(* Logix 5000 project; controller reports 1756-L63 rev 20.15; software revision 20.04; part 37 of 52 *)

        [52].log_data[51].valid := 1, [52].log_data[52].min := -1.6399994, [52].log_data[52].max := -1.4800034, [52].log_data[52].total := -5567.262, [52].log_data[52].time := 3600.0, [52].log_data[52].minminute := 39, [52].log_data[52].valid := 1, [52].log_data[53].min := -1.5600052, [52].log_data[53].max := -1.4199982, [52].log_data[53].total := -5304.3613, [52].log_data[53].time := 3600.0, [52].log_data[53].minminute := 16, [52].log_data[53].valid := 1, [52].log_data[54].time := 3600.0, [52].log_data[54].valid := 1, [52].log_data[55].time := 3600.0, [52].log_data[55].valid := 1, [52].log_data[56].min := 0.16024561, [52].log_data[56].max := 0.16063818, [52].log_data[56].total := 577.39246, [52].log_data[56].time := 3600.0, [52].log_data[56].minminute := 9, [52].log_data[56].valid := 1, [52].log_data[57].min := 0.27864859, [52].log_data[57].max := 0.27904117, [52].log_data[57].total := 1003.6821, [52].log_data[57].time := 3600.0, [52].log_data[57].minminute := 10, [52].log_data[57].maxminute := 2, [52].log_data[57].valid := 1, [52].log_data[58].time := 3600.0, [52].log_data[58].valid := 1, [52].log_data[59].time := 3600.0, [52].log_data[59].valid := 1, [52].log_data[60].valid := 1, [52].log_data[61].valid := 1, [52].log_data[62].valid := 1, [52].log_data[63].valid := 1, [52].log_data[64].valid := 1, [52].log_data[65].valid := 1, [52].log_data[66].valid := 1, [52].log_data[67].valid := 1, [52].log_data[68].valid := 1, [52].log_data[69].valid := 1, [52].log_data[70].valid := 1, [52].log_data[71].valid := 1, [52].log_data[72].valid := 1, [52].log_data[73].valid := 1, [52].log_data[74].valid := 1, [52].log_data[75].valid := 1, [52].log_data[76].valid := 1, [52].log_data[77].valid := 1, [52].log_data[78].valid := 1, [52].log_data[79].valid := 1, [52].log_data[80].valid := 1, [52].log_data[81].valid := 1, [52].log_data[82].valid := 1, [52].log_data[83].valid := 1, [52].log_data[84].valid := 1, [52].log_data[85].valid := 1,
        [52].log_data[86].valid := 1, [52].log_data[87].valid := 1, [52].log_data[88].valid := 1, [52].log_data[89].valid := 1, [52].log_data[90].valid := 1, [52].log_data[91].valid := 1, [52].log_data[92].valid := 1, [52].log_data[93].valid := 1, [52].log_data[94].valid := 1, [52].log_data[95].valid := 1, [52].log_data[96].valid := 1, [52].log_data[97].valid := 1, [52].log_data[98].valid := 1, [52].log_data[99].valid := 1, [52].log_data[100].valid := 1, [52].log_data[101].valid := 1, [52].log_data[102].valid := 1, [52].log_data[103].valid := 1, [52].log_data[104].valid := 1, [52].log_data[105].valid := 1, [52].log_data[106].valid := 1, [52].log_data[107].valid := 1, [52].log_data[108].valid := 1, [52].log_data[109].valid := 1, [52].log_data[110].valid := 1, [52].log_data[111].valid := 1, [52].log_data[112].valid := 1, [52].log_data[113].valid := 1, [52].log_data[114].valid := 1, [52].log_data[115].valid := 1, [52].log_data[116].valid := 1, [52].log_data[117].valid := 1, [52].log_data[118].valid := 1, [52].log_data[119].valid := 1, [52].log_data[120].valid := 1, [52].log_data[121].valid := 1, [52].log_data[122].valid := 1, [52].log_data[123].valid := 1, [52].log_data[124].valid := 1, [52].time.Year := 2023, [52].time.Month := 1, [52].time.Day := 15, [52].time.Hour := 7, [52].time.Minute := 59, [52].time.Second := 59, [53].log_data[0].min := 1.0, [53].log_data[0].max := 1.0, [53].log_data[0].total := 3600.0, [53].log_data[0].time := 3600.0, [53].log_data[0].valid := 1, [53].log_data[1].max := 1.0, [53].log_data[1].total := 543.5, [53].log_data[1].time := 3600.0, [53].log_data[1].maxminute := 32, [53].log_data[1].valid := 1, [53].log_data[2].max := 1.0, [53].log_data[2].total := 540.0, [53].log_data[2].time := 3600.0, [53].log_data[2].maxminute := 32, [53].log_data[2].valid := 1,
        [53].log_data[3].time := 3600.0, [53].log_data[3].valid := 1, [53].log_data[4].time := 3600.0, [53].log_data[4].valid := 1, [53].log_data[5].max := 1.0, [53].log_data[5].total := 221.5, [53].log_data[5].time := 3600.0, [53].log_data[5].maxminute := 33, [53].log_data[5].valid := 1, [53].log_data[6].time := 3600.0, [53].log_data[6].valid := 1, [53].log_data[7].time := 3600.0, [53].log_data[7].valid := 1, [53].log_data[8].max := 1.0, [53].log_data[8].total := 1510.749, [53].log_data[8].time := 3600.0, [53].log_data[8].maxminute := 34, [53].log_data[8].valid := 1, [53].log_data[9].max := 1.0, [53].log_data[9].total := 1507.249, [53].log_data[9].time := 3600.0, [53].log_data[9].maxminute := 34, [53].log_data[9].valid := 1, [53].log_data[10].min := 1.0, [53].log_data[10].max := 1.0, [53].log_data[10].total := 3600.0, [53].log_data[10].time := 3600.0, [53].log_data[10].valid := 1, [53].log_data[11].time := 3600.0, [53].log_data[11].valid := 1, [53].log_data[12].min := 1.0, [53].log_data[12].max := 1.0, [53].log_data[12].total := 3600.0, [53].log_data[12].time := 3600.0, [53].log_data[12].valid := 1, [53].log_data[13].min := 1.0, [53].log_data[13].max := 1.0, [53].log_data[13].total := 3600.0, [53].log_data[13].time := 3600.0, [53].log_data[13].valid := 1, [53].log_data[14].time := 3600.0, [53].log_data[14].valid := 1, [53].log_data[15].time := 3600.0, [53].log_data[15].valid := 1, [53].log_data[16].time := 3600.0, [53].log_data[16].valid := 1, [53].log_data[17].min := 1.0, [53].log_data[17].max := 1.0, [53].log_data[17].total := 3600.0, [53].log_data[17].time := 3600.0, [53].log_data[17].valid := 1, [53].log_data[18].time := 3600.0, [53].log_data[18].valid := 1, [53].log_data[19].time := 3600.0, [53].log_data[19].valid := 1, [53].log_data[20].time := 3600.0, [53].log_data[20].valid := 1, [53].log_data[21].min := 1.0, [53].log_data[21].max := 1.0, [53].log_data[21].total := 3600.0,
        [53].log_data[21].time := 3600.0, [53].log_data[21].valid := 1, [53].log_data[22].time := 3600.0, [53].log_data[22].valid := 1, [53].log_data[23].time := 3600.0, [53].log_data[23].valid := 1, [53].log_data[24].time := 3600.0, [53].log_data[24].valid := 1, [53].log_data[25].time := 3600.0, [53].log_data[25].valid := 1, [53].log_data[26].time := 3600.0, [53].log_data[26].valid := 1, [53].log_data[27].time := 3600.0, [53].log_data[27].valid := 1, [53].log_data[28].time := 3600.0, [53].log_data[28].valid := 1, [53].log_data[29].min := 1.0, [53].log_data[29].max := 1.0, [53].log_data[29].total := 3600.0, [53].log_data[29].time := 3600.0, [53].log_data[29].valid := 1, [53].log_data[30].min := 1.0, [53].log_data[30].max := 1.0, [53].log_data[30].total := 3600.0, [53].log_data[30].time := 3600.0, [53].log_data[30].valid := 1, [53].log_data[31].max := 1.0, [53].log_data[31].total := 543.249, [53].log_data[31].time := 3600.0, [53].log_data[31].maxminute := 43, [53].log_data[31].valid := 1, [53].log_data[32].max := 1.0, [53].log_data[32].total := 783.998, [53].log_data[32].time := 3600.0, [53].log_data[32].maxminute := 34, [53].log_data[32].valid := 1, [53].log_data[33].time := 3600.0, [53].log_data[33].valid := 1, [53].log_data[34].time := 3600.0, [53].log_data[34].valid := 1, [53].log_data[35].max := 1.0, [53].log_data[35].total := 640.49805, [53].log_data[35].time := 3600.0, [53].log_data[35].maxminute := 37, [53].log_data[35].valid := 1, [53].log_data[36].max := 1.0, [53].log_data[36].total := 594.998, [53].log_data[36].time := 3600.0, [53].log_data[36].maxminute := 34, [53].log_data[36].valid := 1, [53].log_data[37].max := 7.248974, [53].log_data[37].total := 3411.01, [53].log_data[37].time := 3600.0, [53].log_data[37].maxminute := 33, [53].log_data[37].valid := 1, [53].log_data[38].time := 3600.0, [53].log_data[38].valid := 1, [53].log_data[39].min := 0.99788606, [53].log_data[39].max := 1.0216767, [53].log_data[39].total := 3646.9153,
        [53].log_data[39].time := 3600.0, [53].log_data[39].minminute := 35, [53].log_data[39].maxminute := 37, [53].log_data[39].valid := 1, [53].log_data[40].min := 7.5687137, [53].log_data[40].max := 7.6019654, [53].log_data[40].total := 27316.076, [53].log_data[40].time := 3600.0, [53].log_data[40].minminute := 7, [53].log_data[40].maxminute := 11, [53].log_data[40].valid := 1, [53].log_data[41].min := 0.025680907, [53].log_data[41].max := 0.045309816, [53].log_data[41].total := 128.45833, [53].log_data[41].time := 3600.0, [53].log_data[41].minminute := 59, [53].log_data[41].maxminute := 29, [53].log_data[41].valid := 1, [53].log_data[42].min := 2.2918782, [53].log_data[42].max := 2.296707, [53].log_data[42].total := 8260.53, [53].log_data[42].time := 3600.0, [53].log_data[42].minminute := 43, [53].log_data[42].maxminute := 41, [53].log_data[42].valid := 1, [53].log_data[43].min := -0.27999878, [53].log_data[43].max := -0.26000214, [53].log_data[43].total := -988.176, [53].log_data[43].time := 3600.0, [53].log_data[43].valid := 1, [53].log_data[44].min := -0.30000305, [53].log_data[44].max := -0.30000305, [53].log_data[44].total := -1080.0911, [53].log_data[44].time := 3600.0, [53].log_data[44].valid := 1, [53].log_data[45].time := 3600.0, [53].log_data[45].valid := 1, [53].log_data[46].time := 3600.0, [53].log_data[46].valid := 1, [53].log_data[47].time := 3600.0, [53].log_data[47].valid := 1, [53].log_data[48].min := 6.6066113, [53].log_data[48].max := 6.9619374, [53].log_data[48].total := 24341.145, [53].log_data[48].time := 3600.0, [53].log_data[48].minminute := 59, [53].log_data[48].maxminute := 39, [53].log_data[48].valid := 1, [53].log_data[49].min := 7.224471, [53].log_data[49].max := 9.765266, [53].log_data[49].total := 32563.492, [53].log_data[49].time := 3600.0, [53].log_data[49].minminute := 55, [53].log_data[49].maxminute := 20, [53].log_data[49].valid := 1, [53].log_data[50].min := 2.061275, [53].log_data[50].max := 2.150784, [53].log_data[50].total := 7565.2534, [53].log_data[50].time := 3600.0, [53].log_data[50].minminute := 37,
        [53].log_data[50].maxminute := 34, [53].log_data[50].valid := 1, [53].log_data[51].time := 3600.0, [53].log_data[51].valid := 1, [53].log_data[52].min := -4.3799973, [53].log_data[52].max := 0.11999512, [53].log_data[52].total := -6630.809, [53].log_data[52].time := 3600.0, [53].log_data[52].minminute := 35, [53].log_data[52].maxminute := 41, [53].log_data[52].valid := 1, [53].log_data[53].min := -3.9399948, [53].log_data[53].max := 0.27999878, [53].log_data[53].total := -5923.6562, [53].log_data[53].time := 3600.0, [53].log_data[53].minminute := 35, [53].log_data[53].maxminute := 58, [53].log_data[53].valid := 1, [53].log_data[54].max := 0.5165, [53].log_data[54].total := 524.9467, [53].log_data[54].time := 3600.0, [53].log_data[54].maxminute := 35, [53].log_data[54].valid := 1, [53].log_data[55].max := 0.5265, [53].log_data[55].total := 486.45926, [53].log_data[55].time := 3600.0, [53].log_data[55].maxminute := 58, [53].log_data[55].valid := 1, [53].log_data[56].min := 0.16016708, [53].log_data[56].max := 0.16059892, [53].log_data[56].total := 577.3497, [53].log_data[56].time := 3600.0, [53].log_data[56].minminute := 43, [53].log_data[56].maxminute := 5, [53].log_data[56].valid := 1, [53].log_data[57].min := 0.27860934, [53].log_data[57].max := 0.27904117, [53].log_data[57].total := 1003.57135, [53].log_data[57].time := 3600.0, [53].log_data[57].minminute := 7, [53].log_data[57].maxminute := 13, [53].log_data[57].valid := 1, [53].log_data[58].time := 3600.0, [53].log_data[58].valid := 1, [53].log_data[59].time := 3600.0, [53].log_data[59].valid := 1, [53].log_data[60].valid := 1, [53].log_data[61].valid := 1, [53].log_data[62].valid := 1, [53].log_data[63].valid := 1, [53].log_data[64].valid := 1, [53].log_data[65].valid := 1, [53].log_data[66].valid := 1, [53].log_data[67].valid := 1, [53].log_data[68].valid := 1, [53].log_data[69].valid := 1, [53].log_data[70].valid := 1, [53].log_data[71].valid := 1, [53].log_data[72].valid := 1, [53].log_data[73].valid := 1,
        [53].log_data[74].valid := 1, [53].log_data[75].valid := 1, [53].log_data[76].valid := 1, [53].log_data[77].valid := 1, [53].log_data[78].valid := 1, [53].log_data[79].valid := 1, [53].log_data[80].valid := 1, [53].log_data[81].valid := 1, [53].log_data[82].valid := 1, [53].log_data[83].valid := 1, [53].log_data[84].valid := 1, [53].log_data[85].valid := 1, [53].log_data[86].valid := 1, [53].log_data[87].valid := 1, [53].log_data[88].valid := 1, [53].log_data[89].valid := 1, [53].log_data[90].valid := 1, [53].log_data[91].valid := 1, [53].log_data[92].valid := 1, [53].log_data[93].valid := 1, [53].log_data[94].valid := 1, [53].log_data[95].valid := 1, [53].log_data[96].valid := 1, [53].log_data[97].valid := 1, [53].log_data[98].valid := 1, [53].log_data[99].valid := 1, [53].log_data[100].valid := 1, [53].log_data[101].valid := 1, [53].log_data[102].valid := 1, [53].log_data[103].valid := 1, [53].log_data[104].valid := 1, [53].log_data[105].valid := 1, [53].log_data[106].valid := 1, [53].log_data[107].valid := 1, [53].log_data[108].valid := 1, [53].log_data[109].valid := 1, [53].log_data[110].valid := 1, [53].log_data[111].valid := 1, [53].log_data[112].valid := 1, [53].log_data[113].valid := 1, [53].log_data[114].valid := 1, [53].log_data[115].valid := 1, [53].log_data[116].valid := 1, [53].log_data[117].valid := 1, [53].log_data[118].valid := 1, [53].log_data[119].valid := 1, [53].log_data[120].valid := 1, [53].log_data[121].valid := 1, [53].log_data[122].valid := 1, [53].log_data[123].valid := 1, [53].log_data[124].valid := 1, [53].time.Year := 2023, [53].time.Month := 1, [53].time.Day := 15, [53].time.Hour := 8, [53].time.Minute := 59, [53].time.Second := 59, [54].log_data[0].min := 1.0, [54].log_data[0].max := 1.0, [54].log_data[0].total := 3600.0,
        [54].log_data[0].time := 3600.0, [54].log_data[0].valid := 1, [54].log_data[1].time := 3600.0, [54].log_data[1].valid := 1, [54].log_data[2].time := 3600.0, [54].log_data[2].valid := 1, [54].log_data[3].time := 3600.0, [54].log_data[3].valid := 1, [54].log_data[4].time := 3600.0, [54].log_data[4].valid := 1, [54].log_data[5].max := 1.0, [54].log_data[5].total := 46.5, [54].log_data[5].time := 3600.0, [54].log_data[5].maxminute := 2, [54].log_data[5].valid := 1, [54].log_data[6].time := 3600.0, [54].log_data[6].valid := 1, [54].log_data[7].time := 3600.0, [54].log_data[7].valid := 1, [54].log_data[8].min := 1.0, [54].log_data[8].max := 1.0, [54].log_data[8].total := 3600.0, [54].log_data[8].time := 3600.0, [54].log_data[8].valid := 1, [54].log_data[9].min := 1.0, [54].log_data[9].max := 1.0, [54].log_data[9].total := 3600.0, [54].log_data[9].time := 3600.0, [54].log_data[9].valid := 1, [54].log_data[10].min := 1.0, [54].log_data[10].max := 1.0, [54].log_data[10].total := 3600.0, [54].log_data[10].time := 3600.0, [54].log_data[10].valid := 1, [54].log_data[11].time := 3600.0, [54].log_data[11].valid := 1, [54].log_data[12].min := 1.0, [54].log_data[12].max := 1.0, [54].log_data[12].total := 3600.0, [54].log_data[12].time := 3600.0, [54].log_data[12].valid := 1, [54].log_data[13].min := 1.0, [54].log_data[13].max := 1.0, [54].log_data[13].total := 3600.0, [54].log_data[13].time := 3600.0, [54].log_data[13].valid := 1, [54].log_data[14].time := 3600.0, [54].log_data[14].valid := 1, [54].log_data[15].time := 3600.0, [54].log_data[15].valid := 1, [54].log_data[16].time := 3600.0, [54].log_data[16].valid := 1, [54].log_data[17].min := 1.0, [54].log_data[17].max := 1.0, [54].log_data[17].total := 3600.0, [54].log_data[17].time := 3600.0, [54].log_data[17].valid := 1, [54].log_data[18].time := 3600.0, [54].log_data[18].valid := 1, [54].log_data[19].time := 3600.0,
        [54].log_data[19].valid := 1, [54].log_data[20].time := 3600.0, [54].log_data[20].valid := 1, [54].log_data[21].min := 1.0, [54].log_data[21].max := 1.0, [54].log_data[21].total := 3600.0, [54].log_data[21].time := 3600.0, [54].log_data[21].valid := 1, [54].log_data[22].time := 3600.0, [54].log_data[22].valid := 1, [54].log_data[23].time := 3600.0, [54].log_data[23].valid := 1, [54].log_data[24].time := 3600.0, [54].log_data[24].valid := 1, [54].log_data[25].time := 3600.0, [54].log_data[25].valid := 1, [54].log_data[26].time := 3600.0, [54].log_data[26].valid := 1, [54].log_data[27].time := 3600.0, [54].log_data[27].valid := 1, [54].log_data[28].time := 3600.0, [54].log_data[28].valid := 1, [54].log_data[29].min := 1.0, [54].log_data[29].max := 1.0, [54].log_data[29].total := 3600.0, [54].log_data[29].time := 3600.0, [54].log_data[29].valid := 1, [54].log_data[30].min := 1.0, [54].log_data[30].max := 1.0, [54].log_data[30].total := 3600.0, [54].log_data[30].time := 3600.0, [54].log_data[30].valid := 1, [54].log_data[31].max := 1.0, [54].log_data[31].total := 1629.998, [54].log_data[31].time := 3600.0, [54].log_data[31].maxminute := 4, [54].log_data[31].valid := 1, [54].log_data[32].max := 1.0, [54].log_data[32].total := 1440.498, [54].log_data[32].time := 3600.0, [54].log_data[32].minminute := 2, [54].log_data[32].valid := 1, [54].log_data[33].time := 3600.0, [54].log_data[33].valid := 1, [54].log_data[34].time := 3600.0, [54].log_data[34].valid := 1, [54].log_data[35].max := 1.0, [54].log_data[35].total := 1532.249, [54].log_data[35].time := 3600.0, [54].log_data[35].minminute := 7, [54].log_data[35].valid := 1, [54].log_data[36].max := 1.0, [54].log_data[36].total := 1626.2471, [54].log_data[36].time := 3600.0, [54].log_data[36].maxminute := 8, [54].log_data[36].valid := 1, [54].log_data[37].time := 3600.0, [54].log_data[37].valid := 1, [54].log_data[38].time := 3600.0, [54].log_data[38].valid := 1,
        [54].log_data[39].min := 0.9956484, [54].log_data[39].max := 1.0202634, [54].log_data[39].total := 3613.4626, [54].log_data[39].time := 3600.0, [54].log_data[39].minminute := 15, [54].log_data[39].maxminute := 2, [54].log_data[39].valid := 1, [54].log_data[40].min := 7.561569, [54].log_data[40].max := 7.603339, [54].log_data[40].total := 27314.873, [54].log_data[40].time := 3600.0, [54].log_data[40].minminute := 48, [54].log_data[40].maxminute := 51, [54].log_data[40].valid := 1, [54].log_data[41].min := 0.022540038, [54].log_data[41].max := 0.03628052, [54].log_data[41].total := 103.08068, [54].log_data[41].time := 3600.0, [54].log_data[41].minminute := 3, [54].log_data[41].maxminute := 37, [54].log_data[41].valid := 1, [54].log_data[42].min := 2.2918782, [54].log_data[42].max := 2.296707, [54].log_data[42].total := 8260.271, [54].log_data[42].time := 3600.0, [54].log_data[42].minminute := 30, [54].log_data[42].maxminute := 36, [54].log_data[42].valid := 1, [54].log_data[43].min := -0.27999878, [54].log_data[43].max := -0.26000214, [54].log_data[43].total := -958.51483, [54].log_data[43].time := 3600.0, [54].log_data[43].valid := 1, [54].log_data[44].min := -0.30000305, [54].log_data[44].max := -0.27999878, [54].log_data[44].total := -1075.2991, [54].log_data[44].time := 3600.0, [54].log_data[44].maxminute := 35, [54].log_data[44].valid := 1, [54].log_data[45].time := 3600.0, [54].log_data[45].valid := 1, [54].log_data[46].time := 3600.0, [54].log_data[46].valid := 1, [54].log_data[47].time := 3600.0, [54].log_data[47].valid := 1, [54].log_data[48].min := 6.585176, [54].log_data[48].max := 6.8080454, [54].log_data[48].total := 24163.797, [54].log_data[48].time := 3600.0, [54].log_data[48].minminute := 2, [54].log_data[48].maxminute := 3, [54].log_data[48].valid := 1, [54].log_data[49].min := 7.171669, [54].log_data[49].max := 9.702061, [54].log_data[49].total := 31267.357, [54].log_data[49].time := 3600.0, [54].log_data[49].minminute := 7, [54].log_data[49].maxminute := 59, [54].log_data[49].valid := 1, [54].log_data[50].min := 2.0161674,
        [54].log_data[50].max := 2.0949588, [54].log_data[50].total := 7409.2114, [54].log_data[50].time := 3600.0, [54].log_data[50].minminute := 59, [54].log_data[50].maxminute := 4, [54].log_data[50].valid := 1, [54].log_data[51].time := 3600.0, [54].log_data[51].valid := 1, [54].log_data[52].min := -2.9400024, [54].log_data[52].max := 0.11999512, [54].log_data[52].total := -7493.728, [54].log_data[52].time := 3600.0, [54].log_data[52].minminute := 25, [54].log_data[52].maxminute := 2, [54].log_data[52].valid := 1, [54].log_data[53].min := -2.5, [54].log_data[53].max := 0.22000122, [54].log_data[53].total := -7034.502, [54].log_data[53].time := 3600.0, [54].log_data[53].minminute := 19, [54].log_data[53].maxminute := 8, [54].log_data[53].valid := 1, [54].log_data[54].max := 0.5245, [54].log_data[54].total := 1217.0215, [54].log_data[54].time := 3600.0, [54].log_data[54].minminute := 2, [54].log_data[54].maxminute := 25, [54].log_data[54].valid := 1, [54].log_data[55].max := 0.533, [54].log_data[55].total := 1254.002, [54].log_data[55].time := 3600.0, [54].log_data[55].minminute := 7, [54].log_data[55].maxminute := 19, [54].log_data[55].valid := 1, [54].log_data[56].min := 0.16012783, [54].log_data[56].max := 0.16059892, [54].log_data[56].total := 577.2283, [54].log_data[56].time := 3600.0, [54].log_data[56].minminute := 17, [54].log_data[56].maxminute := 34, [54].log_data[56].valid := 1, [54].log_data[57].min := 0.27684268, [54].log_data[57].max := 0.2789234, [54].log_data[57].total := 998.60736, [54].log_data[57].time := 3600.0, [54].log_data[57].minminute := 31, [54].log_data[57].valid := 1, [54].log_data[58].time := 3600.0, [54].log_data[58].valid := 1, [54].log_data[59].time := 3600.0, [54].log_data[59].valid := 1, [54].log_data[60].valid := 1, [54].log_data[61].valid := 1, [54].log_data[62].valid := 1, [54].log_data[63].valid := 1, [54].log_data[64].valid := 1, [54].log_data[65].valid := 1, [54].log_data[66].valid := 1, [54].log_data[67].valid := 1, [54].log_data[68].valid := 1,
        [54].log_data[69].valid := 1, [54].log_data[70].valid := 1, [54].log_data[71].valid := 1, [54].log_data[72].valid := 1, [54].log_data[73].valid := 1, [54].log_data[74].valid := 1, [54].log_data[75].valid := 1, [54].log_data[76].valid := 1, [54].log_data[77].valid := 1, [54].log_data[78].valid := 1, [54].log_data[79].valid := 1, [54].log_data[80].valid := 1, [54].log_data[81].valid := 1, [54].log_data[82].valid := 1, [54].log_data[83].valid := 1, [54].log_data[84].valid := 1, [54].log_data[85].valid := 1, [54].log_data[86].valid := 1, [54].log_data[87].valid := 1, [54].log_data[88].valid := 1, [54].log_data[89].valid := 1, [54].log_data[90].valid := 1, [54].log_data[91].valid := 1, [54].log_data[92].valid := 1, [54].log_data[93].valid := 1, [54].log_data[94].valid := 1, [54].log_data[95].valid := 1, [54].log_data[96].valid := 1, [54].log_data[97].valid := 1, [54].log_data[98].valid := 1, [54].log_data[99].valid := 1, [54].log_data[100].valid := 1, [54].log_data[101].valid := 1, [54].log_data[102].valid := 1, [54].log_data[103].valid := 1, [54].log_data[104].valid := 1, [54].log_data[105].valid := 1, [54].log_data[106].valid := 1, [54].log_data[107].valid := 1, [54].log_data[108].valid := 1, [54].log_data[109].valid := 1, [54].log_data[110].valid := 1, [54].log_data[111].valid := 1, [54].log_data[112].valid := 1, [54].log_data[113].valid := 1, [54].log_data[114].valid := 1, [54].log_data[115].valid := 1, [54].log_data[116].valid := 1, [54].log_data[117].valid := 1, [54].log_data[118].valid := 1, [54].log_data[119].valid := 1, [54].log_data[120].valid := 1, [54].log_data[121].valid := 1, [54].log_data[122].valid := 1, [54].log_data[123].valid := 1, [54].log_data[124].valid := 1, [54].time.Year := 2023, [54].time.Month := 1, [54].time.Day := 15, [54].time.Hour := 9,
        [54].time.Minute := 59, [54].time.Second := 59, [55].log_data[0].min := 1.0, [55].log_data[0].max := 1.0, [55].log_data[0].total := 3600.0, [55].log_data[0].time := 3600.0, [55].log_data[0].valid := 1, [55].log_data[1].max := 1.0, [55].log_data[1].total := 546.5, [55].log_data[1].time := 3600.0, [55].log_data[1].maxminute := 12, [55].log_data[1].valid := 1, [55].log_data[2].max := 1.0, [55].log_data[2].total := 543.0, [55].log_data[2].time := 3600.0, [55].log_data[2].maxminute := 12, [55].log_data[2].valid := 1, [55].log_data[3].time := 3600.0, [55].log_data[3].valid := 1, [55].log_data[4].time := 3600.0, [55].log_data[4].valid := 1, [55].log_data[5].max := 1.0, [55].log_data[5].total := 234.0, [55].log_data[5].time := 3600.0, [55].log_data[5].maxminute := 14, [55].log_data[5].valid := 1, [55].log_data[6].time := 3600.0, [55].log_data[6].valid := 1, [55].log_data[7].time := 3600.0, [55].log_data[7].valid := 1, [55].log_data[8].max := 1.0, [55].log_data[8].total := 3158.0, [55].log_data[8].time := 3600.0, [55].log_data[8].minminute := 11, [55].log_data[8].valid := 1, [55].log_data[9].max := 1.0, [55].log_data[9].total := 3154.5, [55].log_data[9].time := 3600.0, [55].log_data[9].minminute := 11, [55].log_data[9].valid := 1, [55].log_data[10].min := 1.0, [55].log_data[10].max := 1.0, [55].log_data[10].total := 3600.0, [55].log_data[10].time := 3600.0, [55].log_data[10].valid := 1, [55].log_data[11].time := 3600.0, [55].log_data[11].valid := 1, [55].log_data[12].min := 1.0, [55].log_data[12].max := 1.0, [55].log_data[12].total := 3600.0, [55].log_data[12].time := 3600.0, [55].log_data[12].valid := 1, [55].log_data[13].min := 1.0, [55].log_data[13].max := 1.0, [55].log_data[13].total := 3600.0, [55].log_data[13].time := 3600.0, [55].log_data[13].valid := 1, [55].log_data[14].time := 3600.0, [55].log_data[14].valid := 1, [55].log_data[15].time := 3600.0,
        [55].log_data[15].valid := 1, [55].log_data[16].time := 3600.0, [55].log_data[16].valid := 1, [55].log_data[17].min := 1.0, [55].log_data[17].max := 1.0, [55].log_data[17].total := 3600.0, [55].log_data[17].time := 3600.0, [55].log_data[17].valid := 1, [55].log_data[18].time := 3600.0, [55].log_data[18].valid := 1, [55].log_data[19].time := 3600.0, [55].log_data[19].valid := 1, [55].log_data[20].time := 3600.0, [55].log_data[20].valid := 1, [55].log_data[21].min := 1.0, [55].log_data[21].max := 1.0, [55].log_data[21].total := 3600.0, [55].log_data[21].time := 3600.0, [55].log_data[21].valid := 1, [55].log_data[22].time := 3600.0, [55].log_data[22].valid := 1, [55].log_data[23].time := 3600.0, [55].log_data[23].valid := 1, [55].log_data[24].time := 3600.0, [55].log_data[24].valid := 1, [55].log_data[25].time := 3600.0, [55].log_data[25].valid := 1, [55].log_data[26].time := 3600.0, [55].log_data[26].valid := 1, [55].log_data[27].time := 3600.0, [55].log_data[27].valid := 1, [55].log_data[28].time := 3600.0, [55].log_data[28].valid := 1, [55].log_data[29].min := 1.0, [55].log_data[29].max := 1.0, [55].log_data[29].total := 3600.0, [55].log_data[29].time := 3600.0, [55].log_data[29].valid := 1, [55].log_data[30].min := 1.0, [55].log_data[30].max := 1.0, [55].log_data[30].total := 3600.0, [55].log_data[30].time := 3600.0, [55].log_data[30].valid := 1, [55].log_data[31].max := 1.0, [55].log_data[31].total := 1324.747, [55].log_data[31].time := 3600.0, [55].log_data[31].maxminute := 7, [55].log_data[31].valid := 1, [55].log_data[32].max := 1.0, [55].log_data[32].total := 1388.998, [55].log_data[32].time := 3600.0, [55].log_data[32].minminute := 5, [55].log_data[32].valid := 1, [55].log_data[33].time := 3600.0, [55].log_data[33].valid := 1, [55].log_data[34].time := 3600.0, [55].log_data[34].valid := 1, [55].log_data[35].max := 1.0, [55].log_data[35].total := 1629.998, [55].log_data[35].time := 3600.0,
        [55].log_data[35].maxminute := 1, [55].log_data[35].valid := 1, [55].log_data[36].max := 1.0, [55].log_data[36].total := 1089.998, [55].log_data[36].time := 3600.0, [55].log_data[36].valid := 1, [55].log_data[37].max := 7.579529, [55].log_data[37].total := 3599.3506, [55].log_data[37].time := 3600.0, [55].log_data[37].maxminute := 14, [55].log_data[37].valid := 1, [55].log_data[38].time := 3600.0, [55].log_data[38].valid := 1, [55].log_data[39].min := 0.997415, [55].log_data[39].max := 1.0214411, [55].log_data[39].total := 3618.071, [55].log_data[39].time := 3600.0, [55].log_data[39].minminute := 56, [55].log_data[39].maxminute := 14, [55].log_data[39].valid := 1, [55].log_data[40].min := 7.5588202, [55].log_data[40].max := 7.6060877, [55].log_data[40].total := 27314.547, [55].log_data[40].time := 3600.0, [55].log_data[40].minminute := 53, [55].log_data[40].maxminute := 57, [55].log_data[40].valid := 1, [55].log_data[41].min := 0.022540038, [55].log_data[41].max := 0.0402063, [55].log_data[41].total := 100.198784, [55].log_data[41].time := 3600.0, [55].log_data[41].minminute := 2, [55].log_data[41].maxminute := 53, [55].log_data[41].valid := 1, [55].log_data[42].min := 2.2916427, [55].log_data[42].max := 2.2965894, [55].log_data[42].total := 8260.112, [55].log_data[42].time := 3600.0, [55].log_data[42].minminute := 25, [55].log_data[42].maxminute := 2, [55].log_data[42].valid := 1, [55].log_data[43].min := -0.26000214, [55].log_data[43].max := -0.26000214, [55].log_data[43].total := -935.9732, [55].log_data[43].time := 3600.0, [55].log_data[43].valid := 1, [55].log_data[44].min := -0.30000305, [55].log_data[44].max := -0.27999878, [55].log_data[44].total := -1017.55457, [55].log_data[44].time := 3600.0, [55].log_data[44].valid := 1, [55].log_data[45].time := 3600.0, [55].log_data[45].valid := 1, [55].log_data[46].time := 3600.0, [55].log_data[46].valid := 1, [55].log_data[47].time := 3600.0, [55].log_data[47].valid := 1, [55].log_data[48].min := 6.573634, [55].log_data[48].max := 6.9666095, [55].log_data[48].total := 24185.111,
        [55].log_data[48].time := 3600.0, [55].log_data[48].minminute := 43, [55].log_data[48].maxminute := 21, [55].log_data[48].valid := 1, [55].log_data[49].min := 7.0474157, [55].log_data[49].max := 9.719335, [55].log_data[49].total := 29908.883, [55].log_data[49].time := 3600.0, [55].log_data[49].minminute := 40, [55].log_data[49].maxminute := 7, [55].log_data[49].valid := 1, [55].log_data[50].min := 1.9992077, [55].log_data[50].max := 2.1516085, [55].log_data[50].total := 7475.81, [55].log_data[50].time := 3600.0, [55].log_data[50].minminute := 11, [55].log_data[50].maxminute := 18, [55].log_data[50].valid := 1, [55].log_data[51].time := 3600.0, [55].log_data[51].valid := 1, [55].log_data[52].min := -4.040001, [55].log_data[52].max := 0.13999939, [55].log_data[52].total := -7179.858, [55].log_data[52].time := 3600.0, [55].log_data[52].minminute := 18, [55].log_data[52].maxminute := 6, [55].log_data[52].valid := 1, [55].log_data[53].min := -3.9399948, [55].log_data[53].max := 0.22000122, [55].log_data[53].total := -6600.5337, [55].log_data[53].time := 3600.0, [55].log_data[53].minminute := 18, [55].log_data[53].valid := 1, [55].log_data[54].max := 0.5775, [55].log_data[54].total := 1074.4722, [55].log_data[54].time := 3600.0, [55].log_data[54].minminute := 5, [55].log_data[54].maxminute := 46, [55].log_data[54].valid := 1, [55].log_data[55].max := 0.522, [55].log_data[55].total := 1079.2233, [55].log_data[55].time := 3600.0, [55].log_data[55].maxminute := 29, [55].log_data[55].valid := 1, [55].log_data[56].min := 0.16012783, [55].log_data[56].max := 0.16055967, [55].log_data[56].total := 577.1176, [55].log_data[56].time := 3600.0, [55].log_data[56].minminute := 41, [55].log_data[56].maxminute := 1, [55].log_data[56].valid := 1, [55].log_data[57].min := 0.27527237, [55].log_data[57].max := 0.2772353, [55].log_data[57].total := 995.83575, [55].log_data[57].time := 3600.0, [55].log_data[57].minminute := 57, [55].log_data[57].maxminute := 1, [55].log_data[57].valid := 1, [55].log_data[58].time := 3600.0, [55].log_data[58].valid := 1,
        [55].log_data[59].time := 3600.0, [55].log_data[59].valid := 1, [55].log_data[60].valid := 1, [55].log_data[61].valid := 1, [55].log_data[62].valid := 1, [55].log_data[63].valid := 1, [55].log_data[64].valid := 1, [55].log_data[65].valid := 1, [55].log_data[66].valid := 1, [55].log_data[67].valid := 1, [55].log_data[68].valid := 1, [55].log_data[69].valid := 1, [55].log_data[70].valid := 1, [55].log_data[71].valid := 1, [55].log_data[72].valid := 1, [55].log_data[73].valid := 1, [55].log_data[74].valid := 1, [55].log_data[75].valid := 1, [55].log_data[76].valid := 1, [55].log_data[77].valid := 1, [55].log_data[78].valid := 1, [55].log_data[79].valid := 1, [55].log_data[80].valid := 1, [55].log_data[81].valid := 1, [55].log_data[82].valid := 1, [55].log_data[83].valid := 1, [55].log_data[84].valid := 1, [55].log_data[85].valid := 1, [55].log_data[86].valid := 1, [55].log_data[87].valid := 1, [55].log_data[88].valid := 1, [55].log_data[89].valid := 1, [55].log_data[90].valid := 1, [55].log_data[91].valid := 1, [55].log_data[92].valid := 1, [55].log_data[93].valid := 1, [55].log_data[94].valid := 1, [55].log_data[95].valid := 1, [55].log_data[96].valid := 1, [55].log_data[97].valid := 1, [55].log_data[98].valid := 1, [55].log_data[99].valid := 1, [55].log_data[100].valid := 1, [55].log_data[101].valid := 1, [55].log_data[102].valid := 1, [55].log_data[103].valid := 1, [55].log_data[104].valid := 1, [55].log_data[105].valid := 1, [55].log_data[106].valid := 1, [55].log_data[107].valid := 1, [55].log_data[108].valid := 1, [55].log_data[109].valid := 1, [55].log_data[110].valid := 1, [55].log_data[111].valid := 1, [55].log_data[112].valid := 1, [55].log_data[113].valid := 1, [55].log_data[114].valid := 1, [55].log_data[115].valid := 1, [55].log_data[116].valid := 1, [55].log_data[117].valid := 1,
        [55].log_data[118].valid := 1, [55].log_data[119].valid := 1, [55].log_data[120].valid := 1, [55].log_data[121].valid := 1, [55].log_data[122].valid := 1, [55].log_data[123].valid := 1, [55].log_data[124].valid := 1, [55].time.Year := 2023, [55].time.Month := 1, [55].time.Day := 15, [55].time.Hour := 10, [55].time.Minute := 59, [55].time.Second := 59, [56].log_data[0].min := 1.0, [56].log_data[0].max := 1.0, [56].log_data[0].total := 3599.5, [56].log_data[0].time := 3599.5, [56].log_data[0].valid := 1, [56].log_data[1].max := 1.0, [56].log_data[1].total := 574.0, [56].log_data[1].time := 3599.5, [56].log_data[1].maxminute := 25, [56].log_data[1].valid := 1, [56].log_data[2].max := 1.0, [56].log_data[2].total := 570.5, [56].log_data[2].time := 3599.5, [56].log_data[2].maxminute := 25, [56].log_data[2].valid := 1, [56].log_data[3].time := 3599.5, [56].log_data[3].valid := 1, [56].log_data[4].time := 3599.5, [56].log_data[4].valid := 1, [56].log_data[5].max := 1.0, [56].log_data[5].total := 252.0, [56].log_data[5].time := 3599.5, [56].log_data[5].maxminute := 27, [56].log_data[5].valid := 1, [56].log_data[6].time := 3599.5, [56].log_data[6].valid := 1, [56].log_data[7].time := 3599.5, [56].log_data[7].valid := 1, [56].log_data[8].min := 1.0, [56].log_data[8].max := 1.0, [56].log_data[8].total := 3599.5, [56].log_data[8].time := 3599.5, [56].log_data[8].valid := 1, [56].log_data[9].min := 1.0, [56].log_data[9].max := 1.0, [56].log_data[9].total := 3599.5, [56].log_data[9].time := 3599.5, [56].log_data[9].valid := 1, [56].log_data[10].min := 1.0, [56].log_data[10].max := 1.0, [56].log_data[10].total := 3599.5, [56].log_data[10].time := 3599.5, [56].log_data[10].valid := 1, [56].log_data[11].time := 3599.5, [56].log_data[11].valid := 1, [56].log_data[12].min := 1.0, [56].log_data[12].max := 1.0,
        [56].log_data[12].total := 3599.5, [56].log_data[12].time := 3599.5, [56].log_data[12].valid := 1, [56].log_data[13].min := 1.0, [56].log_data[13].max := 1.0, [56].log_data[13].total := 3599.5, [56].log_data[13].time := 3599.5, [56].log_data[13].valid := 1, [56].log_data[14].time := 3599.5, [56].log_data[14].valid := 1, [56].log_data[15].time := 3599.5, [56].log_data[15].valid := 1, [56].log_data[16].time := 3599.5, [56].log_data[16].valid := 1, [56].log_data[17].min := 1.0, [56].log_data[17].max := 1.0, [56].log_data[17].total := 3599.5, [56].log_data[17].time := 3599.5, [56].log_data[17].valid := 1, [56].log_data[18].time := 3599.5, [56].log_data[18].valid := 1, [56].log_data[19].time := 3599.5, [56].log_data[19].valid := 1, [56].log_data[20].time := 3599.5, [56].log_data[20].valid := 1, [56].log_data[21].min := 1.0, [56].log_data[21].max := 1.0, [56].log_data[21].total := 3599.5, [56].log_data[21].time := 3599.5, [56].log_data[21].valid := 1, [56].log_data[22].time := 3599.5, [56].log_data[22].valid := 1, [56].log_data[23].time := 3599.5, [56].log_data[23].valid := 1, [56].log_data[24].time := 3599.5, [56].log_data[24].valid := 1, [56].log_data[25].time := 3599.5, [56].log_data[25].valid := 1, [56].log_data[26].time := 3599.5, [56].log_data[26].valid := 1, [56].log_data[27].time := 3599.5, [56].log_data[27].valid := 1, [56].log_data[28].time := 3599.5, [56].log_data[28].valid := 1, [56].log_data[29].min := 1.0, [56].log_data[29].max := 1.0, [56].log_data[29].total := 3599.5, [56].log_data[29].time := 3599.5, [56].log_data[29].valid := 1, [56].log_data[30].min := 1.0, [56].log_data[30].max := 1.0, [56].log_data[30].total := 3599.5, [56].log_data[30].time := 3599.5, [56].log_data[30].valid := 1, [56].log_data[31].max := 1.0, [56].log_data[31].total := 1629.7471, [56].log_data[31].time := 3599.5, [56].log_data[31].maxminute := 7, [56].log_data[31].valid := 1, [56].log_data[32].max := 1.0,
        [56].log_data[32].total := 1442.249, [56].log_data[32].time := 3599.5, [56].log_data[32].minminute := 5, [56].log_data[32].valid := 1, [56].log_data[33].time := 3599.5, [56].log_data[33].valid := 1, [56].log_data[34].time := 3599.5, [56].log_data[34].valid := 1, [56].log_data[35].max := 1.0, [56].log_data[35].total := 1473.749, [56].log_data[35].time := 3599.5, [56].log_data[35].maxminute := 11, [56].log_data[35].valid := 1, [56].log_data[36].max := 1.0, [56].log_data[36].total := 1629.998, [56].log_data[36].time := 3599.5, [56].log_data[36].valid := 1, [56].log_data[37].max := 7.346335, [56].log_data[37].total := 3671.0361, [56].log_data[37].time := 3599.5, [56].log_data[37].maxminute := 27, [56].log_data[37].valid := 1, [56].log_data[38].time := 3599.5, [56].log_data[38].valid := 1, [56].log_data[39].min := 0.99623734, [56].log_data[39].max := 1.0232078, [56].log_data[39].total := 3617.8582, [56].log_data[39].time := 3599.5, [56].log_data[39].minminute := 29, [56].log_data[39].maxminute := 31, [56].log_data[39].valid := 1, [56].log_data[40].min := 7.5758586, [56].log_data[40].max := 7.5961943, [56].log_data[40].total := 27315.29, [56].log_data[40].time := 3599.5, [56].log_data[40].minminute := 6, [56].log_data[40].maxminute := 10, [56].log_data[40].valid := 1, [56].log_data[41].min := 0.025680907, [56].log_data[41].max := 0.043543212, [56].log_data[41].total := 122.82056, [56].log_data[41].time := 3599.5, [56].log_data[41].minminute := 56, [56].log_data[41].maxminute := 26, [56].log_data[41].valid := 1, [56].log_data[42].min := 2.291407, [56].log_data[42].max := 2.2964714, [56].log_data[42].total := 8258.96, [56].log_data[42].time := 3599.5, [56].log_data[42].minminute := 20, [56].log_data[42].maxminute := 4, [56].log_data[42].valid := 1, [56].log_data[43].min := -0.26000214, [56].log_data[43].max := -0.26000214, [56].log_data[43].total := -935.8432, [56].log_data[43].time := 3599.5, [56].log_data[43].valid := 1, [56].log_data[44].min := -0.30000305, [56].log_data[44].max := -0.27999878, [56].log_data[44].total := -1023.11255,
        [56].log_data[44].time := 3599.5, [56].log_data[44].valid := 1, [56].log_data[45].time := 3599.5, [56].log_data[45].valid := 1, [56].log_data[46].time := 3599.5, [56].log_data[46].valid := 1, [56].log_data[47].time := 3599.5, [56].log_data[47].valid := 1, [56].log_data[48].min := 6.57968, [56].log_data[48].max := 6.945174, [56].log_data[48].total := 24245.596, [56].log_data[48].time := 3599.5, [56].log_data[48].minminute := 56, [56].log_data[48].maxminute := 29, [56].log_data[48].valid := 1, [56].log_data[49].min := 6.9688993, [56].log_data[49].max := 9.635517, [56].log_data[49].total := 30506.39, [56].log_data[49].time := 3599.5, [56].log_data[49].minminute := 52, [56].log_data[49].maxminute := 27, [56].log_data[49].valid := 1, [56].log_data[50].min := 2.0234694, [56].log_data[50].max := 2.1391244, [56].log_data[50].total := 7499.3022, [56].log_data[50].time := 3599.5, [56].log_data[50].minminute := 27, [56].log_data[50].maxminute := 34, [56].log_data[50].valid := 1, [56].log_data[51].time := 3599.5, [56].log_data[51].valid := 1, [56].log_data[52].min := -3.040001, [56].log_data[52].max := 0.13999939, [56].log_data[52].total := -7567.2183, [56].log_data[52].time := 3599.5, [56].log_data[52].minminute := 49, [56].log_data[52].maxminute := 27, [56].log_data[52].valid := 1, [56].log_data[53].min := -2.7000046, [56].log_data[53].max := 0.2400055, [56].log_data[53].total := -7021.4707, [56].log_data[53].time := 3599.5, [56].log_data[53].minminute := 43, [56].log_data[53].maxminute := 42, [56].log_data[53].valid := 1, [56].log_data[54].max := 0.55799997, [56].log_data[54].total := 1219.9869, [56].log_data[54].time := 3599.5, [56].log_data[54].minminute := 5, [56].log_data[54].maxminute := 49, [56].log_data[54].valid := 1, [56].log_data[55].max := 0.55149996, [56].log_data[55].total := 1230.2097, [56].log_data[55].time := 3599.5, [56].log_data[55].maxminute := 43, [56].log_data[55].valid := 1, [56].log_data[56].min := 0.16008857, [56].log_data[56].max := 0.1605204, [56].log_data[56].total := 576.9246, [56].log_data[56].time := 3599.5,
        [56].log_data[56].minminute := 54, [56].log_data[56].valid := 1, [56].log_data[57].min := 0.27433017, [56].log_data[57].max := 0.27562568, [56].log_data[57].total := 990.9707, [56].log_data[57].time := 3599.5, [56].log_data[57].minminute := 59, [56].log_data[57].valid := 1, [56].log_data[58].time := 3599.5, [56].log_data[58].valid := 1, [56].log_data[59].time := 3599.5, [56].log_data[59].valid := 1, [56].log_data[60].valid := 1, [56].log_data[61].valid := 1, [56].log_data[62].valid := 1, [56].log_data[63].valid := 1, [56].log_data[64].valid := 1, [56].log_data[65].valid := 1, [56].log_data[66].valid := 1, [56].log_data[67].valid := 1, [56].log_data[68].valid := 1, [56].log_data[69].valid := 1, [56].log_data[70].valid := 1, [56].log_data[71].valid := 1, [56].log_data[72].valid := 1, [56].log_data[73].valid := 1, [56].log_data[74].valid := 1, [56].log_data[75].valid := 1, [56].log_data[76].valid := 1, [56].log_data[77].valid := 1, [56].log_data[78].valid := 1, [56].log_data[79].valid := 1, [56].log_data[80].valid := 1, [56].log_data[81].valid := 1, [56].log_data[82].valid := 1, [56].log_data[83].valid := 1, [56].log_data[84].valid := 1, [56].log_data[85].valid := 1, [56].log_data[86].valid := 1, [56].log_data[87].valid := 1, [56].log_data[88].valid := 1, [56].log_data[89].valid := 1, [56].log_data[90].valid := 1, [56].log_data[91].valid := 1, [56].log_data[92].valid := 1, [56].log_data[93].valid := 1, [56].log_data[94].valid := 1, [56].log_data[95].valid := 1, [56].log_data[96].valid := 1, [56].log_data[97].valid := 1, [56].log_data[98].valid := 1, [56].log_data[99].valid := 1, [56].log_data[100].valid := 1, [56].log_data[101].valid := 1, [56].log_data[102].valid := 1, [56].log_data[103].valid := 1, [56].log_data[104].valid := 1, [56].log_data[105].valid := 1, [56].log_data[106].valid := 1, [56].log_data[107].valid := 1,
        [56].log_data[108].valid := 1, [56].log_data[109].valid := 1, [56].log_data[110].valid := 1, [56].log_data[111].valid := 1, [56].log_data[112].valid := 1, [56].log_data[113].valid := 1, [56].log_data[114].valid := 1, [56].log_data[115].valid := 1, [56].log_data[116].valid := 1, [56].log_data[117].valid := 1, [56].log_data[118].valid := 1, [56].log_data[119].valid := 1, [56].log_data[120].valid := 1, [56].log_data[121].valid := 1, [56].log_data[122].valid := 1, [56].log_data[123].valid := 1, [56].log_data[124].valid := 1, [56].time.Year := 2023, [56].time.Month := 1, [56].time.Day := 15, [56].time.Hour := 11, [56].time.Minute := 59, [56].time.Second := 59, [57].log_data[0].min := 1.0, [57].log_data[0].max := 1.0, [57].log_data[0].total := 3600.0, [57].log_data[0].time := 3600.0, [57].log_data[0].valid := 1, [57].log_data[1].max := 1.0, [57].log_data[1].total := 555.5, [57].log_data[1].time := 3600.0, [57].log_data[1].maxminute := 37, [57].log_data[1].valid := 1, [57].log_data[2].max := 1.0, [57].log_data[2].total := 552.0, [57].log_data[2].time := 3600.0, [57].log_data[2].maxminute := 37, [57].log_data[2].valid := 1, [57].log_data[3].time := 3600.0, [57].log_data[3].valid := 1, [57].log_data[4].time := 3600.0, [57].log_data[4].valid := 1, [57].log_data[5].max := 1.0, [57].log_data[5].total := 246.0, [57].log_data[5].time := 3600.0, [57].log_data[5].maxminute := 39, [57].log_data[5].valid := 1, [57].log_data[6].time := 3600.0, [57].log_data[6].valid := 1, [57].log_data[7].time := 3600.0, [57].log_data[7].valid := 1, [57].log_data[8].min := 1.0, [57].log_data[8].max := 1.0, [57].log_data[8].total := 3600.0, [57].log_data[8].time := 3600.0, [57].log_data[8].valid := 1, [57].log_data[9].min := 1.0, [57].log_data[9].max := 1.0, [57].log_data[9].total := 3600.0, [57].log_data[9].time := 3600.0,
        [57].log_data[9].valid := 1, [57].log_data[10].min := 1.0, [57].log_data[10].max := 1.0, [57].log_data[10].total := 3600.0, [57].log_data[10].time := 3600.0, [57].log_data[10].valid := 1, [57].log_data[11].time := 3600.0, [57].log_data[11].valid := 1, [57].log_data[12].min := 1.0, [57].log_data[12].max := 1.0, [57].log_data[12].total := 3600.0, [57].log_data[12].time := 3600.0, [57].log_data[12].valid := 1, [57].log_data[13].min := 1.0, [57].log_data[13].max := 1.0, [57].log_data[13].total := 3600.0, [57].log_data[13].time := 3600.0, [57].log_data[13].valid := 1, [57].log_data[14].time := 3600.0, [57].log_data[14].valid := 1, [57].log_data[15].time := 3600.0, [57].log_data[15].valid := 1, [57].log_data[16].time := 3600.0, [57].log_data[16].valid := 1, [57].log_data[17].min := 1.0, [57].log_data[17].max := 1.0, [57].log_data[17].total := 3600.0, [57].log_data[17].time := 3600.0, [57].log_data[17].valid := 1, [57].log_data[18].time := 3600.0, [57].log_data[18].valid := 1, [57].log_data[19].time := 3600.0, [57].log_data[19].valid := 1, [57].log_data[20].time := 3600.0, [57].log_data[20].valid := 1, [57].log_data[21].min := 1.0, [57].log_data[21].max := 1.0, [57].log_data[21].total := 3600.0, [57].log_data[21].time := 3600.0, [57].log_data[21].valid := 1, [57].log_data[22].time := 3600.0, [57].log_data[22].valid := 1, [57].log_data[23].time := 3600.0, [57].log_data[23].valid := 1, [57].log_data[24].time := 3600.0, [57].log_data[24].valid := 1, [57].log_data[25].time := 3600.0, [57].log_data[25].valid := 1, [57].log_data[26].time := 3600.0, [57].log_data[26].valid := 1, [57].log_data[27].time := 3600.0, [57].log_data[27].valid := 1, [57].log_data[28].time := 3600.0, [57].log_data[28].valid := 1, [57].log_data[29].min := 1.0, [57].log_data[29].max := 1.0, [57].log_data[29].total := 3600.0, [57].log_data[29].time := 3600.0, [57].log_data[29].valid := 1, [57].log_data[30].min := 1.0,
        [57].log_data[30].max := 1.0, [57].log_data[30].total := 3600.0, [57].log_data[30].time := 3600.0, [57].log_data[30].valid := 1, [57].log_data[31].max := 1.0, [57].log_data[31].total := 1527.2471, [57].log_data[31].time := 3600.0, [57].log_data[31].maxminute := 10, [57].log_data[31].valid := 1, [57].log_data[32].max := 1.0, [57].log_data[32].total := 1629.998, [57].log_data[32].time := 3600.0, [57].log_data[32].valid := 1, [57].log_data[33].time := 3600.0, [57].log_data[33].valid := 1, [57].log_data[34].time := 3600.0, [57].log_data[34].valid := 1, [57].log_data[35].max := 1.0, [57].log_data[35].total := 1440.7471, [57].log_data[35].time := 3600.0, [57].log_data[35].minminute := 2, [57].log_data[35].valid := 1, [57].log_data[36].max := 1.0, [57].log_data[36].total := 1629.7471, [57].log_data[36].time := 3600.0, [57].log_data[36].maxminute := 4, [57].log_data[36].valid := 1, [57].log_data[37].max := 7.5991583, [57].log_data[37].total := 3665.0671, [57].log_data[37].time := 3600.0, [57].log_data[37].maxminute := 39, [57].log_data[37].valid := 1, [57].log_data[38].time := 3600.0, [57].log_data[38].valid := 1, [57].log_data[39].min := 0.995884, [57].log_data[39].max := 1.0219122, [57].log_data[39].total := 3617.047, [57].log_data[39].time := 3600.0, [57].log_data[39].minminute := 11, [57].log_data[39].maxminute := 44, [57].log_data[39].valid := 1, [57].log_data[40].min := 7.5714617, [57].log_data[40].max := 7.5961943, [57].log_data[40].total := 27316.074, [57].log_data[40].time := 3600.0, [57].log_data[40].minminute := 35, [57].log_data[40].maxminute := 7, [57].log_data[40].valid := 1, [57].log_data[41].min := 0.02273633, [57].log_data[41].max := 0.033139892, [57].log_data[41].total := 91.76312, [57].log_data[41].time := 3600.0, [57].log_data[41].minminute := 11, [57].log_data[41].maxminute := 18, [57].log_data[41].valid := 1, [57].log_data[42].min := 2.2918782, [57].log_data[42].max := 2.2965894, [57].log_data[42].total := 8260.124, [57].log_data[42].time := 3600.0, [57].log_data[42].minminute := 51,
        [57].log_data[42].maxminute := 19, [57].log_data[42].valid := 1, [57].log_data[43].min := -0.27999878, [57].log_data[43].max := -0.26000214, [57].log_data[43].total := -938.2722, [57].log_data[43].time := 3600.0, [57].log_data[43].minminute := 15, [57].log_data[43].valid := 1, [57].log_data[44].min := -0.30000305, [57].log_data[44].max := -0.27999878, [57].log_data[44].total := -1069.6058, [57].log_data[44].time := 3600.0, [57].log_data[44].valid := 1, [57].log_data[45].time := 3600.0, [57].log_data[45].valid := 1, [57].log_data[46].time := 3600.0, [57].log_data[46].valid := 1, [57].log_data[47].time := 3600.0, [57].log_data[47].valid := 1, [57].log_data[48].min := 6.6082597, [57].log_data[48].max := 6.980624, [57].log_data[48].total := 24351.37, [57].log_data[48].time := 3600.0, [57].log_data[48].maxminute := 45, [57].log_data[48].valid := 1, [57].log_data[49].min := 7.071953, [57].log_data[49].max := 9.62531, [57].log_data[49].total := 30890.484, [57].log_data[49].time := 3600.0, [57].log_data[49].maxminute := 39, [57].log_data[49].valid := 1, [57].log_data[50].min := 2.0490265, [57].log_data[50].max := 2.1657412, [57].log_data[50].total := 7568.1777, [57].log_data[50].time := 3600.0, [57].log_data[50].minminute := 39, [57].log_data[50].maxminute := 46, [57].log_data[50].valid := 1, [57].log_data[51].time := 3600.0, [57].log_data[51].valid := 1, [57].log_data[52].min := -2.880005, [57].log_data[52].max := 0.13999939, [57].log_data[52].total := -7763.1943, [57].log_data[52].time := 3600.0, [57].log_data[52].minminute := 10, [57].log_data[52].maxminute := 9, [57].log_data[52].valid := 1, [57].log_data[53].min := -2.5200043, [57].log_data[53].max := 0.2400055, [57].log_data[53].total := -6941.8887, [57].log_data[53].time := 3600.0, [57].log_data[53].minminute := 56, [57].log_data[53].maxminute := 3, [57].log_data[53].valid := 1, [57].log_data[54].max := 0.518, [57].log_data[54].total := 1251.6619, [57].log_data[54].time := 3600.0, [57].log_data[54].maxminute := 10, [57].log_data[54].valid := 1, [57].log_data[55].max := 0.5395,
        [57].log_data[55].total := 1217.4039, [57].log_data[55].time := 3600.0, [57].log_data[55].minminute := 2, [57].log_data[55].maxminute := 56, [57].log_data[55].valid := 1, [57].log_data[56].min := 0.1599708, [57].log_data[56].max := 0.1605204, [57].log_data[56].total := 576.769, [57].log_data[56].time := 3600.0, [57].log_data[56].minminute := 39, [57].log_data[56].maxminute := 20, [57].log_data[56].valid := 1, [57].log_data[57].min := 0.2731132, [57].log_data[57].max := 0.27444795, [57].log_data[57].total := 984.2539, [57].log_data[57].time := 3600.0, [57].log_data[57].minminute := 40, [57].log_data[57].valid := 1, [57].log_data[58].time := 3600.0, [57].log_data[58].valid := 1, [57].log_data[59].time := 3600.0, [57].log_data[59].valid := 1, [57].log_data[60].valid := 1, [57].log_data[61].valid := 1, [57].log_data[62].valid := 1, [57].log_data[63].valid := 1, [57].log_data[64].valid := 1, [57].log_data[65].valid := 1, [57].log_data[66].valid := 1, [57].log_data[67].valid := 1, [57].log_data[68].valid := 1, [57].log_data[69].valid := 1, [57].log_data[70].valid := 1, [57].log_data[71].valid := 1, [57].log_data[72].valid := 1, [57].log_data[73].valid := 1, [57].log_data[74].valid := 1, [57].log_data[75].valid := 1, [57].log_data[76].valid := 1, [57].log_data[77].valid := 1, [57].log_data[78].valid := 1, [57].log_data[79].valid := 1, [57].log_data[80].valid := 1, [57].log_data[81].valid := 1, [57].log_data[82].valid := 1, [57].log_data[83].valid := 1, [57].log_data[84].valid := 1, [57].log_data[85].valid := 1, [57].log_data[86].valid := 1, [57].log_data[87].valid := 1, [57].log_data[88].valid := 1, [57].log_data[89].valid := 1, [57].log_data[90].valid := 1, [57].log_data[91].valid := 1, [57].log_data[92].valid := 1, [57].log_data[93].valid := 1, [57].log_data[94].valid := 1, [57].log_data[95].valid := 1, [57].log_data[96].valid := 1, [57].log_data[97].valid := 1,
        [57].log_data[98].valid := 1, [57].log_data[99].valid := 1, [57].log_data[100].valid := 1, [57].log_data[101].valid := 1, [57].log_data[102].valid := 1, [57].log_data[103].valid := 1, [57].log_data[104].valid := 1, [57].log_data[105].valid := 1, [57].log_data[106].valid := 1, [57].log_data[107].valid := 1, [57].log_data[108].valid := 1, [57].log_data[109].valid := 1, [57].log_data[110].valid := 1, [57].log_data[111].valid := 1, [57].log_data[112].valid := 1, [57].log_data[113].valid := 1, [57].log_data[114].valid := 1, [57].log_data[115].valid := 1, [57].log_data[116].valid := 1, [57].log_data[117].valid := 1, [57].log_data[118].valid := 1, [57].log_data[119].valid := 1, [57].log_data[120].valid := 1, [57].log_data[121].valid := 1, [57].log_data[122].valid := 1, [57].log_data[123].valid := 1, [57].log_data[124].valid := 1, [57].time.Year := 2023, [57].time.Month := 1, [57].time.Day := 15, [57].time.Hour := 12, [57].time.Minute := 59, [57].time.Second := 59, [58].log_data[0].min := 1.0, [58].log_data[0].max := 1.0, [58].log_data[0].total := 3600.0, [58].log_data[0].time := 3600.0, [58].log_data[0].valid := 1, [58].log_data[1].max := 1.0, [58].log_data[1].total := 567.0, [58].log_data[1].time := 3600.0, [58].log_data[1].maxminute := 50, [58].log_data[1].valid := 1, [58].log_data[2].max := 1.0, [58].log_data[2].total := 563.5, [58].log_data[2].time := 3600.0, [58].log_data[2].maxminute := 50, [58].log_data[2].valid := 1, [58].log_data[3].time := 3600.0, [58].log_data[3].valid := 1, [58].log_data[4].time := 3600.0, [58].log_data[4].valid := 1, [58].log_data[5].max := 1.0, [58].log_data[5].total := 241.0, [58].log_data[5].time := 3600.0, [58].log_data[5].maxminute := 52, [58].log_data[5].valid := 1, [58].log_data[6].time := 3600.0, [58].log_data[6].valid := 1, [58].log_data[7].time := 3600.0,
        [58].log_data[7].valid := 1, [58].log_data[8].min := 1.0, [58].log_data[8].max := 1.0, [58].log_data[8].total := 3600.0, [58].log_data[8].time := 3600.0, [58].log_data[8].valid := 1, [58].log_data[9].min := 1.0, [58].log_data[9].max := 1.0, [58].log_data[9].total := 3600.0, [58].log_data[9].time := 3600.0, [58].log_data[9].valid := 1, [58].log_data[10].min := 1.0, [58].log_data[10].max := 1.0, [58].log_data[10].total := 3600.0, [58].log_data[10].time := 3600.0, [58].log_data[10].valid := 1, [58].log_data[11].time := 3600.0, [58].log_data[11].valid := 1, [58].log_data[12].min := 1.0, [58].log_data[12].max := 1.0, [58].log_data[12].total := 3600.0, [58].log_data[12].time := 3600.0, [58].log_data[12].valid := 1, [58].log_data[13].min := 1.0, [58].log_data[13].max := 1.0, [58].log_data[13].total := 3600.0, [58].log_data[13].time := 3600.0, [58].log_data[13].valid := 1, [58].log_data[14].time := 3600.0, [58].log_data[14].valid := 1, [58].log_data[15].time := 3600.0, [58].log_data[15].valid := 1, [58].log_data[16].time := 3600.0, [58].log_data[16].valid := 1, [58].log_data[17].min := 1.0, [58].log_data[17].max := 1.0, [58].log_data[17].total := 3600.0, [58].log_data[17].time := 3600.0, [58].log_data[17].valid := 1, [58].log_data[18].time := 3600.0, [58].log_data[18].valid := 1, [58].log_data[19].time := 3600.0, [58].log_data[19].valid := 1, [58].log_data[20].time := 3600.0, [58].log_data[20].valid := 1, [58].log_data[21].min := 1.0, [58].log_data[21].max := 1.0, [58].log_data[21].total := 3600.0, [58].log_data[21].time := 3600.0, [58].log_data[21].valid := 1, [58].log_data[22].time := 3600.0, [58].log_data[22].valid := 1, [58].log_data[23].time := 3600.0, [58].log_data[23].valid := 1, [58].log_data[24].time := 3600.0, [58].log_data[24].valid := 1, [58].log_data[25].time := 3600.0, [58].log_data[25].valid := 1, [58].log_data[26].time := 3600.0, [58].log_data[26].valid := 1,
        [58].log_data[27].time := 3600.0, [58].log_data[27].valid := 1, [58].log_data[28].time := 3600.0, [58].log_data[28].valid := 1, [58].log_data[29].min := 1.0, [58].log_data[29].max := 1.0, [58].log_data[29].total := 3600.0, [58].log_data[29].time := 3600.0, [58].log_data[29].valid := 1, [58].log_data[30].min := 1.0, [58].log_data[30].max := 1.0, [58].log_data[30].total := 3600.0, [58].log_data[30].time := 3600.0, [58].log_data[30].valid := 1, [58].log_data[31].max := 1.0, [58].log_data[31].total := 1440.7471, [58].log_data[31].time := 3600.0, [58].log_data[31].minminute := 1, [58].log_data[31].valid := 1, [58].log_data[32].max := 1.0, [58].log_data[32].total := 1629.998, [58].log_data[32].time := 3600.0, [58].log_data[32].maxminute := 3, [58].log_data[32].valid := 1, [58].log_data[33].time := 3600.0, [58].log_data[33].valid := 1, [58].log_data[34].time := 3600.0, [58].log_data[34].valid := 1, [58].log_data[35].max := 1.0, [58].log_data[35].total := 1440.7471, [58].log_data[35].time := 3600.0, [58].log_data[35].minminute := 5, [58].log_data[35].valid := 1, [58].log_data[36].max := 1.0, [58].log_data[36].total := 1629.7471, [58].log_data[36].time := 3600.0, [58].log_data[36].maxminute := 7, [58].log_data[36].valid := 1, [58].log_data[37].max := 7.3906965, [58].log_data[37].total := 3634.8633, [58].log_data[37].time := 3600.0, [58].log_data[37].maxminute := 51, [58].log_data[37].valid := 1, [58].log_data[38].time := 3600.0, [58].log_data[38].valid := 1, [58].log_data[39].min := 0.9968262, [58].log_data[39].max := 1.0219122, [58].log_data[39].total := 3616.709, [58].log_data[39].time := 3600.0, [58].log_data[39].minminute := 43, [58].log_data[39].maxminute := 56, [58].log_data[39].valid := 1, [58].log_data[40].min := 7.5645914, [58].log_data[40].max := 7.5950956, [58].log_data[40].total := 27315.557, [58].log_data[40].time := 3600.0, [58].log_data[40].minminute := 56, [58].log_data[40].maxminute := 59, [58].log_data[40].valid := 1, [58].log_data[41].min := 0.02273633,
        [58].log_data[41].max := 0.0384397, [58].log_data[41].total := 111.63304, [58].log_data[41].time := 3600.0, [58].log_data[41].maxminute := 38, [58].log_data[41].valid := 1, [58].log_data[42].min := 2.2916427, [58].log_data[42].max := 2.2965894, [58].log_data[42].total := 8260.084, [58].log_data[42].time := 3600.0, [58].log_data[42].minminute := 58, [58].log_data[42].maxminute := 49, [58].log_data[42].valid := 1, [58].log_data[43].min := -0.27999878, [58].log_data[43].max := -0.26000214, [58].log_data[43].total := -952.6892, [58].log_data[43].time := 3600.0, [58].log_data[43].valid := 1, [58].log_data[44].min := -0.30000305, [58].log_data[44].max := -0.30000305, [58].log_data[44].total := -1080.0911, [58].log_data[44].time := 3600.0, [58].log_data[44].valid := 1, [58].log_data[45].time := 3600.0, [58].log_data[45].valid := 1, [58].log_data[46].time := 3600.0, [58].log_data[46].valid := 1, [58].log_data[47].time := 3600.0, [58].log_data[47].valid := 1, [58].log_data[48].min := 6.5810537, [58].log_data[48].max := 6.9547925, [58].log_data[48].total := 24254.494, [58].log_data[48].time := 3600.0, [58].log_data[48].minminute := 10, [58].log_data[48].maxminute := 55, [58].log_data[48].valid := 1, [58].log_data[49].min := 6.984014, [58].log_data[49].max := 9.652792, [58].log_data[49].total := 30723.432, [58].log_data[49].time := 3600.0, [58].log_data[49].minminute := 2, [58].log_data[49].maxminute := 53, [58].log_data[49].valid := 1, [58].log_data[50].min := 2.076468, [58].log_data[50].max := 2.1877651, [58].log_data[50].total := 7621.2593, [58].log_data[50].time := 3600.0, [58].log_data[50].minminute := 52, [58].log_data[50].maxminute := 59, [58].log_data[50].valid := 1, [58].log_data[51].time := 3600.0, [58].log_data[51].valid := 1, [58].log_data[52].min := -2.9000015, [58].log_data[52].max := 0.11999512, [58].log_data[52].total := -7536.673, [58].log_data[52].time := 3600.0, [58].log_data[52].minminute := 13, [58].log_data[52].maxminute := 1, [58].log_data[52].valid := 1, [58].log_data[53].min := -2.5200043, [58].log_data[53].max := 0.22000122,
        [58].log_data[53].total := -7002.238, [58].log_data[53].time := 3600.0, [58].log_data[53].minminute := 28, [58].log_data[53].maxminute := 7, [58].log_data[53].valid := 1, [58].log_data[54].max := 0.5215, [58].log_data[54].total := 1217.1891, [58].log_data[54].time := 3600.0, [58].log_data[54].minminute := 1, [58].log_data[54].maxminute := 13, [58].log_data[54].valid := 1, [58].log_data[55].max := 0.52099997, [58].log_data[55].total := 1217.9204, [58].log_data[55].time := 3600.0, [58].log_data[55].minminute := 5, [58].log_data[55].maxminute := 17, [58].log_data[55].valid := 1, [58].log_data[56].min := 0.15993154, [58].log_data[56].max := 0.16044189, [58].log_data[56].total := 576.5848, [58].log_data[56].time := 3600.0, [58].log_data[56].minminute := 1, [58].log_data[56].maxminute := 7, [58].log_data[56].valid := 1, [58].log_data[57].min := 0.27111098, [58].log_data[57].max := 0.27358428, [58].log_data[57].total := 978.31226, [58].log_data[57].time := 3600.0, [58].log_data[57].minminute := 56, [58].log_data[57].valid := 1, [58].log_data[58].time := 3600.0, [58].log_data[58].valid := 1, [58].log_data[59].time := 3600.0, [58].log_data[59].valid := 1, [58].log_data[60].valid := 1, [58].log_data[61].valid := 1, [58].log_data[62].valid := 1, [58].log_data[63].valid := 1, [58].log_data[64].valid := 1, [58].log_data[65].valid := 1, [58].log_data[66].valid := 1, [58].log_data[67].valid := 1, [58].log_data[68].valid := 1, [58].log_data[69].valid := 1, [58].log_data[70].valid := 1, [58].log_data[71].valid := 1, [58].log_data[72].valid := 1, [58].log_data[73].valid := 1, [58].log_data[74].valid := 1, [58].log_data[75].valid := 1, [58].log_data[76].valid := 1, [58].log_data[77].valid := 1, [58].log_data[78].valid := 1, [58].log_data[79].valid := 1, [58].log_data[80].valid := 1, [58].log_data[81].valid := 1, [58].log_data[82].valid := 1, [58].log_data[83].valid := 1, [58].log_data[84].valid := 1, [58].log_data[85].valid := 1,
        [58].log_data[86].valid := 1, [58].log_data[87].valid := 1, [58].log_data[88].valid := 1, [58].log_data[89].valid := 1, [58].log_data[90].valid := 1, [58].log_data[91].valid := 1, [58].log_data[92].valid := 1, [58].log_data[93].valid := 1, [58].log_data[94].valid := 1, [58].log_data[95].valid := 1, [58].log_data[96].valid := 1, [58].log_data[97].valid := 1, [58].log_data[98].valid := 1, [58].log_data[99].valid := 1, [58].log_data[100].valid := 1, [58].log_data[101].valid := 1, [58].log_data[102].valid := 1, [58].log_data[103].valid := 1, [58].log_data[104].valid := 1, [58].log_data[105].valid := 1, [58].log_data[106].valid := 1, [58].log_data[107].valid := 1, [58].log_data[108].valid := 1, [58].log_data[109].valid := 1, [58].log_data[110].valid := 1, [58].log_data[111].valid := 1, [58].log_data[112].valid := 1, [58].log_data[113].valid := 1, [58].log_data[114].valid := 1, [58].log_data[115].valid := 1, [58].log_data[116].valid := 1, [58].log_data[117].valid := 1, [58].log_data[118].valid := 1, [58].log_data[119].valid := 1, [58].log_data[120].valid := 1, [58].log_data[121].valid := 1, [58].log_data[122].valid := 1, [58].log_data[123].valid := 1, [58].log_data[124].valid := 1, [58].time.Year := 2023, [58].time.Month := 1, [58].time.Day := 15, [58].time.Hour := 13, [58].time.Minute := 59, [58].time.Second := 59, [59].log_data[0].min := 1.0, [59].log_data[0].max := 1.0, [59].log_data[0].total := 3600.0, [59].log_data[0].time := 3600.0, [59].log_data[0].valid := 1, [59].log_data[1].time := 3600.0, [59].log_data[1].valid := 1, [59].log_data[2].time := 3600.0, [59].log_data[2].valid := 1, [59].log_data[3].time := 3600.0, [59].log_data[3].valid := 1, [59].log_data[4].time := 3600.0, [59].log_data[4].valid := 1, [59].log_data[5].time := 3600.0, [59].log_data[5].valid := 1,
        [59].log_data[6].time := 3600.0, [59].log_data[6].valid := 1, [59].log_data[7].time := 3600.0, [59].log_data[7].valid := 1, [59].log_data[8].min := 1.0, [59].log_data[8].max := 1.0, [59].log_data[8].total := 3600.0, [59].log_data[8].time := 3600.0, [59].log_data[8].valid := 1, [59].log_data[9].min := 1.0, [59].log_data[9].max := 1.0, [59].log_data[9].total := 3600.0, [59].log_data[9].time := 3600.0, [59].log_data[9].valid := 1, [59].log_data[10].min := 1.0, [59].log_data[10].max := 1.0, [59].log_data[10].total := 3600.0, [59].log_data[10].time := 3600.0, [59].log_data[10].valid := 1, [59].log_data[11].time := 3600.0, [59].log_data[11].valid := 1, [59].log_data[12].min := 1.0, [59].log_data[12].max := 1.0, [59].log_data[12].total := 3600.0, [59].log_data[12].time := 3600.0, [59].log_data[12].valid := 1, [59].log_data[13].min := 1.0, [59].log_data[13].max := 1.0, [59].log_data[13].total := 3600.0, [59].log_data[13].time := 3600.0, [59].log_data[13].valid := 1, [59].log_data[14].time := 3600.0, [59].log_data[14].valid := 1, [59].log_data[15].time := 3600.0, [59].log_data[15].valid := 1, [59].log_data[16].time := 3600.0, [59].log_data[16].valid := 1, [59].log_data[17].min := 1.0, [59].log_data[17].max := 1.0, [59].log_data[17].total := 3600.0, [59].log_data[17].time := 3600.0, [59].log_data[17].valid := 1, [59].log_data[18].time := 3600.0, [59].log_data[18].valid := 1, [59].log_data[19].time := 3600.0, [59].log_data[19].valid := 1, [59].log_data[20].time := 3600.0, [59].log_data[20].valid := 1, [59].log_data[21].min := 1.0, [59].log_data[21].max := 1.0, [59].log_data[21].total := 3600.0, [59].log_data[21].time := 3600.0, [59].log_data[21].valid := 1, [59].log_data[22].time := 3600.0, [59].log_data[22].valid := 1, [59].log_data[23].time := 3600.0, [59].log_data[23].valid := 1, [59].log_data[24].time := 3600.0, [59].log_data[24].valid := 1, [59].log_data[25].time := 3600.0,
        [59].log_data[25].valid := 1, [59].log_data[26].time := 3600.0, [59].log_data[26].valid := 1, [59].log_data[27].time := 3600.0, [59].log_data[27].valid := 1, [59].log_data[28].time := 3600.0, [59].log_data[28].valid := 1, [59].log_data[29].min := 1.0, [59].log_data[29].max := 1.0, [59].log_data[29].total := 3600.0, [59].log_data[29].time := 3600.0, [59].log_data[29].valid := 1, [59].log_data[30].min := 1.0, [59].log_data[30].max := 1.0, [59].log_data[30].total := 3600.0, [59].log_data[30].time := 3600.0, [59].log_data[30].valid := 1, [59].log_data[31].max := 1.0, [59].log_data[31].total := 1440.7471, [59].log_data[31].time := 3600.0, [59].log_data[31].minminute := 4, [59].log_data[31].valid := 1, [59].log_data[32].max := 1.0, [59].log_data[32].total := 1629.7471, [59].log_data[32].time := 3600.0, [59].log_data[32].maxminute := 6, [59].log_data[32].valid := 1, [59].log_data[33].time := 3600.0, [59].log_data[33].valid := 1, [59].log_data[34].time := 3600.0, [59].log_data[34].valid := 1, [59].log_data[35].max := 1.0, [59].log_data[35].total := 1620.498, [59].log_data[35].time := 3600.0, [59].log_data[35].minminute := 8, [59].log_data[35].valid := 1, [59].log_data[36].max := 1.0, [59].log_data[36].total := 1538.2471, [59].log_data[36].time := 3600.0, [59].log_data[36].maxminute := 10, [59].log_data[36].valid := 1, [59].log_data[37].time := 3600.0, [59].log_data[37].valid := 1, [59].log_data[38].time := 3600.0, [59].log_data[38].valid := 1, [59].log_data[39].min := 0.99788606, [59].log_data[39].max := 1.0093104, [59].log_data[39].total := 3617.053, [59].log_data[39].time := 3600.0, [59].log_data[39].minminute := 27, [59].log_data[39].maxminute := 28, [59].log_data[39].valid := 1, [59].log_data[40].min := 7.563218, [59].log_data[40].max := 7.603614, [59].log_data[40].total := 27322.234, [59].log_data[40].time := 3600.0, [59].log_data[40].minminute := 52, [59].log_data[40].maxminute := 54, [59].log_data[40].valid := 1, [59].log_data[41].min := 0.02273633,
        [59].log_data[41].max := 0.04158032, [59].log_data[41].total := 108.002365, [59].log_data[41].time := 3600.0, [59].log_data[41].minminute := 1, [59].log_data[41].maxminute := 49, [59].log_data[41].valid := 1, [59].log_data[42].min := 2.2916427, [59].log_data[42].max := 2.296707, [59].log_data[42].total := 8260.244, [59].log_data[42].time := 3600.0, [59].log_data[42].minminute := 2, [59].log_data[42].maxminute := 36, [59].log_data[42].valid := 1, [59].log_data[43].min := -0.27999878, [59].log_data[43].max := -0.26000214, [59].log_data[43].total := -986.17163, [59].log_data[43].time := 3600.0, [59].log_data[43].valid := 1, [59].log_data[44].min := -0.3199997, [59].log_data[44].max := -0.30000305, [59].log_data[44].total := -1080.2156, [59].log_data[44].time := 3600.0, [59].log_data[44].minminute := 27, [59].log_data[44].valid := 1, [59].log_data[45].time := 3600.0, [59].log_data[45].valid := 1, [59].log_data[46].time := 3600.0, [59].log_data[46].valid := 1, [59].log_data[47].time := 3600.0, [59].log_data[47].valid := 1, [59].log_data[48].min := 6.5824285, [59].log_data[48].max := 6.8808694, [59].log_data[48].total := 24202.1, [59].log_data[48].time := 3600.0, [59].log_data[48].minminute := 24, [59].log_data[48].valid := 1, [59].log_data[49].min := 7.0238614, [59].log_data[49].max := 9.5854645, [59].log_data[49].total := 29606.55, [59].log_data[49].time := 3600.0, [59].log_data[49].minminute := 22, [59].log_data[49].maxminute := 59, [59].log_data[49].valid := 1, [59].log_data[50].min := 2.104145, [59].log_data[50].max := 2.1878831, [59].log_data[50].total := 7731.9097, [59].log_data[50].time := 3600.0, [59].log_data[50].minminute := 59, [59].log_data[50].valid := 1, [59].log_data[51].time := 3600.0, [59].log_data[51].valid := 1, [59].log_data[52].min := -2.9400024, [59].log_data[52].max := 0.11999512, [59].log_data[52].total := -7591.1646, [59].log_data[52].time := 3600.0, [59].log_data[52].minminute := 59, [59].log_data[52].maxminute := 4, [59].log_data[52].valid := 1, [59].log_data[53].min := -2.6600037, [59].log_data[53].max := 0.27999878,
        [59].log_data[53].total := -7289.749, [59].log_data[53].time := 3600.0, [59].log_data[53].minminute := 20, [59].log_data[53].maxminute := 31, [59].log_data[53].valid := 1, [59].log_data[54].max := 0.52099997, [59].log_data[54].total := 1217.1096, [59].log_data[54].time := 3600.0, [59].log_data[54].minminute := 4, [59].log_data[54].maxminute := 38, [59].log_data[54].valid := 1, [59].log_data[55].max := 0.5475, [59].log_data[55].total := 1253.6866, [59].log_data[55].time := 3600.0, [59].log_data[55].minminute := 8, [59].log_data[55].maxminute := 21, [59].log_data[55].valid := 1, [59].log_data[56].min := 0.15993154, [59].log_data[56].max := 0.16036338, [59].log_data[56].total := 576.4856, [59].log_data[56].time := 3600.0, [59].log_data[56].minminute := 29, [59].log_data[56].valid := 1, [59].log_data[57].min := 0.2693444, [59].log_data[57].max := 0.27154282, [59].log_data[57].total := 973.0487, [59].log_data[57].time := 3600.0, [59].log_data[57].minminute := 38, [59].log_data[57].maxminute := 3, [59].log_data[57].valid := 1, [59].log_data[58].time := 3600.0, [59].log_data[58].valid := 1, [59].log_data[59].time := 3600.0, [59].log_data[59].valid := 1, [59].log_data[60].valid := 1, [59].log_data[61].valid := 1, [59].log_data[62].valid := 1, [59].log_data[63].valid := 1, [59].log_data[64].valid := 1, [59].log_data[65].valid := 1, [59].log_data[66].valid := 1, [59].log_data[67].valid := 1, [59].log_data[68].valid := 1, [59].log_data[69].valid := 1, [59].log_data[70].valid := 1, [59].log_data[71].valid := 1, [59].log_data[72].valid := 1, [59].log_data[73].valid := 1, [59].log_data[74].valid := 1, [59].log_data[75].valid := 1, [59].log_data[76].valid := 1, [59].log_data[77].valid := 1, [59].log_data[78].valid := 1, [59].log_data[79].valid := 1, [59].log_data[80].valid := 1, [59].log_data[81].valid := 1, [59].log_data[82].valid := 1, [59].log_data[83].valid := 1, [59].log_data[84].valid := 1, [59].log_data[85].valid := 1,
        [59].log_data[86].valid := 1, [59].log_data[87].valid := 1, [59].log_data[88].valid := 1, [59].log_data[89].valid := 1, [59].log_data[90].valid := 1, [59].log_data[91].valid := 1, [59].log_data[92].valid := 1, [59].log_data[93].valid := 1, [59].log_data[94].valid := 1, [59].log_data[95].valid := 1, [59].log_data[96].valid := 1, [59].log_data[97].valid := 1, [59].log_data[98].valid := 1, [59].log_data[99].valid := 1, [59].log_data[100].valid := 1, [59].log_data[101].valid := 1, [59].log_data[102].valid := 1, [59].log_data[103].valid := 1, [59].log_data[104].valid := 1, [59].log_data[105].valid := 1, [59].log_data[106].valid := 1, [59].log_data[107].valid := 1, [59].log_data[108].valid := 1, [59].log_data[109].valid := 1, [59].log_data[110].valid := 1, [59].log_data[111].valid := 1, [59].log_data[112].valid := 1, [59].log_data[113].valid := 1, [59].log_data[114].valid := 1, [59].log_data[115].valid := 1, [59].log_data[116].valid := 1, [59].log_data[117].valid := 1, [59].log_data[118].valid := 1, [59].log_data[119].valid := 1, [59].log_data[120].valid := 1, [59].log_data[121].valid := 1, [59].log_data[122].valid := 1, [59].log_data[123].valid := 1, [59].log_data[124].valid := 1, [59].time.Year := 2023, [59].time.Month := 1, [59].time.Day := 15, [59].time.Hour := 14, [59].time.Minute := 59, [59].time.Second := 59, [60].log_data[0].min := 1.0, [60].log_data[0].max := 1.0, [60].log_data[0].total := 3600.0, [60].log_data[0].time := 3600.0, [60].log_data[0].valid := 1, [60].log_data[1].max := 1.0, [60].log_data[1].total := 552.5, [60].log_data[1].time := 3600.0, [60].log_data[1].maxminute := 3, [60].log_data[1].valid := 1, [60].log_data[2].max := 1.0, [60].log_data[2].total := 549.0, [60].log_data[2].time := 3600.0, [60].log_data[2].maxminute := 3, [60].log_data[2].valid := 1,
        [60].log_data[3].time := 3600.0, [60].log_data[3].valid := 1, [60].log_data[4].time := 3600.0, [60].log_data[4].valid := 1, [60].log_data[5].max := 1.0, [60].log_data[5].total := 236.5, [60].log_data[5].time := 3600.0, [60].log_data[5].maxminute := 5, [60].log_data[5].valid := 1, [60].log_data[6].time := 3600.0, [60].log_data[6].valid := 1, [60].log_data[7].time := 3600.0, [60].log_data[7].valid := 1, [60].log_data[8].min := 1.0, [60].log_data[8].max := 1.0, [60].log_data[8].total := 3600.0, [60].log_data[8].time := 3600.0, [60].log_data[8].valid := 1, [60].log_data[9].min := 1.0, [60].log_data[9].max := 1.0, [60].log_data[9].total := 3600.0, [60].log_data[9].time := 3600.0, [60].log_data[9].valid := 1, [60].log_data[10].min := 1.0, [60].log_data[10].max := 1.0, [60].log_data[10].total := 3600.0, [60].log_data[10].time := 3600.0, [60].log_data[10].valid := 1, [60].log_data[11].time := 3600.0, [60].log_data[11].valid := 1, [60].log_data[12].min := 1.0, [60].log_data[12].max := 1.0, [60].log_data[12].total := 3600.0, [60].log_data[12].time := 3600.0, [60].log_data[12].valid := 1, [60].log_data[13].min := 1.0, [60].log_data[13].max := 1.0, [60].log_data[13].total := 3600.0, [60].log_data[13].time := 3600.0, [60].log_data[13].valid := 1, [60].log_data[14].time := 3600.0, [60].log_data[14].valid := 1, [60].log_data[15].time := 3600.0, [60].log_data[15].valid := 1, [60].log_data[16].time := 3600.0, [60].log_data[16].valid := 1, [60].log_data[17].min := 1.0, [60].log_data[17].max := 1.0, [60].log_data[17].total := 3600.0, [60].log_data[17].time := 3600.0, [60].log_data[17].valid := 1, [60].log_data[18].time := 3600.0, [60].log_data[18].valid := 1, [60].log_data[19].time := 3600.0, [60].log_data[19].valid := 1, [60].log_data[20].time := 3600.0, [60].log_data[20].valid := 1, [60].log_data[21].min := 1.0, [60].log_data[21].max := 1.0, [60].log_data[21].total := 3600.0,
        [60].log_data[21].time := 3600.0, [60].log_data[21].valid := 1, [60].log_data[22].time := 3600.0, [60].log_data[22].valid := 1, [60].log_data[23].time := 3600.0, [60].log_data[23].valid := 1, [60].log_data[24].time := 3600.0, [60].log_data[24].valid := 1, [60].log_data[25].time := 3600.0, [60].log_data[25].valid := 1, [60].log_data[26].time := 3600.0, [60].log_data[26].valid := 1, [60].log_data[27].time := 3600.0, [60].log_data[27].valid := 1, [60].log_data[28].time := 3600.0, [60].log_data[28].valid := 1, [60].log_data[29].min := 1.0, [60].log_data[29].max := 1.0, [60].log_data[29].total := 3600.0, [60].log_data[29].time := 3600.0, [60].log_data[29].valid := 1, [60].log_data[30].min := 1.0, [60].log_data[30].max := 1.0, [60].log_data[30].total := 3600.0, [60].log_data[30].time := 3600.0, [60].log_data[30].valid := 1, [60].log_data[31].max := 1.0, [60].log_data[31].total := 1566.998, [60].log_data[31].time := 3600.0, [60].log_data[31].minminute := 8, [60].log_data[31].valid := 1, [60].log_data[32].max := 1.0, [60].log_data[32].total := 1592.249, [60].log_data[32].time := 3600.0, [60].log_data[32].maxminute := 9, [60].log_data[32].valid := 1, [60].log_data[33].time := 3600.0, [60].log_data[33].valid := 1, [60].log_data[34].time := 3600.0, [60].log_data[34].valid := 1, [60].log_data[35].max := 1.0, [60].log_data[35].total := 1629.998, [60].log_data[35].time := 3600.0, [60].log_data[35].maxminute := 2, [60].log_data[35].valid := 1, [60].log_data[36].max := 1.0, [60].log_data[36].total := 1440.2471, [60].log_data[36].time := 3600.0, [60].log_data[36].minminute := 1, [60].log_data[36].valid := 1, [60].log_data[37].max := 7.570107, [60].log_data[37].total := 3621.6538, [60].log_data[37].time := 3600.0, [60].log_data[37].maxminute := 4, [60].log_data[37].valid := 1, [60].log_data[38].time := 3600.0, [60].log_data[38].valid := 1, [60].log_data[39].min := 0.9983573, [60].log_data[39].max := 1.0221478, [60].log_data[39].total := 3625.5813,
        [60].log_data[39].time := 3600.0, [60].log_data[39].minminute := 7, [60].log_data[39].maxminute := 9, [60].log_data[39].valid := 1, [60].log_data[40].min := 7.5703626, [60].log_data[40].max := 7.597843, [60].log_data[40].total := 27320.377, [60].log_data[40].time := 3600.0, [60].log_data[40].minminute := 17, [60].log_data[40].maxminute := 34, [60].log_data[40].valid := 1, [60].log_data[41].min := 0.024895508, [60].log_data[41].max := 0.04570239, [60].log_data[41].total := 129.43713, [60].log_data[41].time := 3600.0, [60].log_data[41].minminute := 59, [60].log_data[41].maxminute := 20, [60].log_data[41].valid := 1, [60].log_data[42].min := 2.2912893, [60].log_data[42].max := 2.296707, [60].log_data[42].total := 8260.318, [60].log_data[42].time := 3600.0, [60].log_data[42].minminute := 14, [60].log_data[42].maxminute := 51, [60].log_data[42].valid := 1, [60].log_data[43].min := -0.27999878, [60].log_data[43].max := -0.26000214, [60].log_data[43].total := -1007.4615, [60].log_data[43].time := 3600.0, [60].log_data[43].valid := 1, [60].log_data[44].min := -0.3199997, [60].log_data[44].max := -0.30000305, [60].log_data[44].total := -1091.5457, [60].log_data[44].time := 3600.0, [60].log_data[44].valid := 1, [60].log_data[45].time := 3600.0, [60].log_data[45].valid := 1, [60].log_data[46].time := 3600.0, [60].log_data[46].valid := 1, [60].log_data[47].time := 3600.0, [60].log_data[47].valid := 1, [60].log_data[48].min := 6.590947, [60].log_data[48].max := 6.9251137, [60].log_data[48].total := 24244.402, [60].log_data[48].time := 3600.0, [60].log_data[48].minminute := 37, [60].log_data[48].maxminute := 7, [60].log_data[48].valid := 1, [60].log_data[49].min := 7.0381904, [60].log_data[49].max := 9.646708, [60].log_data[49].total := 29660.879, [60].log_data[49].time := 3600.0, [60].log_data[49].minminute := 30, [60].log_data[49].maxminute := 5, [60].log_data[49].valid := 1, [60].log_data[50].min := 2.0968432, [60].log_data[50].max := 2.2047248, [60].log_data[50].total := 7797.1426, [60].log_data[50].time := 3600.0, [60].log_data[50].minminute := 5,
        [60].log_data[50].maxminute := 12, [60].log_data[50].valid := 1, [60].log_data[51].time := 3600.0, [60].log_data[51].valid := 1, [60].log_data[52].min := -2.880005, [60].log_data[52].max := 0.11999512, [60].log_data[52].total := -7823.42, [60].log_data[52].time := 3600.0, [60].log_data[52].minminute := 20, [60].log_data[52].maxminute := 8, [60].log_data[52].valid := 1, [60].log_data[53].min := -2.5, [60].log_data[53].max := 0.27999878, [60].log_data[53].total := -7059.904, [60].log_data[53].time := 3600.0, [60].log_data[53].minminute := 56, [60].log_data[53].maxminute := 2, [60].log_data[53].valid := 1, [60].log_data[54].max := 0.5315, [60].log_data[54].total := 1254.5413, [60].log_data[54].time := 3600.0, [60].log_data[54].minminute := 8, [60].log_data[54].maxminute := 20, [60].log_data[54].valid := 1, [60].log_data[55].max := 0.52900004, [60].log_data[55].total := 1217.0195, [60].log_data[55].time := 3600.0, [60].log_data[55].minminute := 1, [60].log_data[55].maxminute := 55, [60].log_data[55].valid := 1, [60].log_data[56].min := 0.15993154, [60].log_data[56].max := 0.16032413, [60].log_data[56].total := 576.34125, [60].log_data[56].time := 3600.0, [60].log_data[56].minminute := 11, [60].log_data[56].valid := 1, [60].log_data[57].min := 0.26797032, [60].log_data[57].max := 0.2696977, [60].log_data[57].total := 968.4547, [60].log_data[57].time := 3600.0, [60].log_data[57].minminute := 45, [60].log_data[57].maxminute := 3, [60].log_data[57].valid := 1, [60].log_data[58].time := 3600.0, [60].log_data[58].valid := 1, [60].log_data[59].time := 3600.0, [60].log_data[59].valid := 1, [60].log_data[60].valid := 1, [60].log_data[61].valid := 1, [60].log_data[62].valid := 1, [60].log_data[63].valid := 1, [60].log_data[64].valid := 1, [60].log_data[65].valid := 1, [60].log_data[66].valid := 1, [60].log_data[67].valid := 1, [60].log_data[68].valid := 1, [60].log_data[69].valid := 1, [60].log_data[70].valid := 1, [60].log_data[71].valid := 1, [60].log_data[72].valid := 1,
        [60].log_data[73].valid := 1, [60].log_data[74].valid := 1, [60].log_data[75].valid := 1, [60].log_data[76].valid := 1, [60].log_data[77].valid := 1, [60].log_data[78].valid := 1, [60].log_data[79].valid := 1, [60].log_data[80].valid := 1, [60].log_data[81].valid := 1, [60].log_data[82].valid := 1, [60].log_data[83].valid := 1, [60].log_data[84].valid := 1, [60].log_data[85].valid := 1, [60].log_data[86].valid := 1, [60].log_data[87].valid := 1, [60].log_data[88].valid := 1, [60].log_data[89].valid := 1, [60].log_data[90].valid := 1, [60].log_data[91].valid := 1, [60].log_data[92].valid := 1, [60].log_data[93].valid := 1, [60].log_data[94].valid := 1, [60].log_data[95].valid := 1, [60].log_data[96].valid := 1, [60].log_data[97].valid := 1, [60].log_data[98].valid := 1, [60].log_data[99].valid := 1, [60].log_data[100].valid := 1, [60].log_data[101].valid := 1, [60].log_data[102].valid := 1, [60].log_data[103].valid := 1, [60].log_data[104].valid := 1, [60].log_data[105].valid := 1, [60].log_data[106].valid := 1, [60].log_data[107].valid := 1, [60].log_data[108].valid := 1, [60].log_data[109].valid := 1, [60].log_data[110].valid := 1, [60].log_data[111].valid := 1, [60].log_data[112].valid := 1, [60].log_data[113].valid := 1, [60].log_data[114].valid := 1, [60].log_data[115].valid := 1, [60].log_data[116].valid := 1, [60].log_data[117].valid := 1, [60].log_data[118].valid := 1, [60].log_data[119].valid := 1, [60].log_data[120].valid := 1, [60].log_data[121].valid := 1, [60].log_data[122].valid := 1, [60].log_data[123].valid := 1, [60].log_data[124].valid := 1, [60].time.Year := 2023, [60].time.Month := 1, [60].time.Day := 15, [60].time.Hour := 15, [60].time.Minute := 59, [60].time.Second := 59, [61].log_data[0].min := 1.0, [61].log_data[0].max := 1.0,
        [61].log_data[0].total := 3600.0, [61].log_data[0].time := 3600.0, [61].log_data[0].valid := 1, [61].log_data[1].max := 1.0, [61].log_data[1].total := 564.0, [61].log_data[1].time := 3600.0, [61].log_data[1].maxminute := 19, [61].log_data[1].valid := 1, [61].log_data[2].max := 1.0, [61].log_data[2].total := 560.5, [61].log_data[2].time := 3600.0, [61].log_data[2].maxminute := 19, [61].log_data[2].valid := 1, [61].log_data[3].time := 3600.0, [61].log_data[3].valid := 1, [61].log_data[4].time := 3600.0, [61].log_data[4].valid := 1, [61].log_data[5].max := 1.0, [61].log_data[5].total := 249.0, [61].log_data[5].time := 3600.0, [61].log_data[5].maxminute := 21, [61].log_data[5].valid := 1, [61].log_data[6].time := 3600.0, [61].log_data[6].valid := 1, [61].log_data[7].time := 3600.0, [61].log_data[7].valid := 1, [61].log_data[8].min := 1.0, [61].log_data[8].max := 1.0, [61].log_data[8].total := 3600.0, [61].log_data[8].time := 3600.0, [61].log_data[8].valid := 1, [61].log_data[9].min := 1.0, [61].log_data[9].max := 1.0, [61].log_data[9].total := 3600.0, [61].log_data[9].time := 3600.0, [61].log_data[9].valid := 1, [61].log_data[10].min := 1.0, [61].log_data[10].max := 1.0, [61].log_data[10].total := 3600.0, [61].log_data[10].time := 3600.0, [61].log_data[10].valid := 1, [61].log_data[11].time := 3600.0, [61].log_data[11].valid := 1, [61].log_data[12].min := 1.0, [61].log_data[12].max := 1.0, [61].log_data[12].total := 3600.0, [61].log_data[12].time := 3600.0, [61].log_data[12].valid := 1, [61].log_data[13].min := 1.0, [61].log_data[13].max := 1.0, [61].log_data[13].total := 3600.0, [61].log_data[13].time := 3600.0, [61].log_data[13].valid := 1, [61].log_data[14].time := 3600.0, [61].log_data[14].valid := 1, [61].log_data[15].time := 3600.0, [61].log_data[15].valid := 1, [61].log_data[16].time := 3600.0, [61].log_data[16].valid := 1, [61].log_data[17].min := 1.0,
        [61].log_data[17].max := 1.0, [61].log_data[17].total := 3600.0, [61].log_data[17].time := 3600.0, [61].log_data[17].valid := 1, [61].log_data[18].time := 3600.0, [61].log_data[18].valid := 1, [61].log_data[19].time := 3600.0, [61].log_data[19].valid := 1, [61].log_data[20].time := 3600.0, [61].log_data[20].valid := 1, [61].log_data[21].min := 1.0, [61].log_data[21].max := 1.0, [61].log_data[21].total := 3600.0, [61].log_data[21].time := 3600.0, [61].log_data[21].valid := 1, [61].log_data[22].time := 3600.0, [61].log_data[22].valid := 1, [61].log_data[23].time := 3600.0, [61].log_data[23].valid := 1, [61].log_data[24].time := 3600.0, [61].log_data[24].valid := 1, [61].log_data[25].time := 3600.0, [61].log_data[25].valid := 1, [61].log_data[26].time := 3600.0, [61].log_data[26].valid := 1, [61].log_data[27].time := 3600.0, [61].log_data[27].valid := 1, [61].log_data[28].time := 3600.0, [61].log_data[28].valid := 1, [61].log_data[29].min := 1.0, [61].log_data[29].max := 1.0, [61].log_data[29].total := 3600.0, [61].log_data[29].time := 3600.0, [61].log_data[29].valid := 1, [61].log_data[30].min := 1.0, [61].log_data[30].max := 1.0, [61].log_data[30].total := 3600.0, [61].log_data[30].time := 3600.0, [61].log_data[30].valid := 1, [61].log_data[31].max := 1.0, [61].log_data[31].total := 1629.998, [61].log_data[31].time := 3600.0, [61].log_data[31].maxminute := 2, [61].log_data[31].valid := 1, [61].log_data[32].max := 1.0, [61].log_data[32].total := 1441.5, [61].log_data[32].time := 3600.0, [61].log_data[32].valid := 1, [61].log_data[33].time := 3600.0, [61].log_data[33].valid := 1, [61].log_data[34].time := 3600.0, [61].log_data[34].valid := 1, [61].log_data[35].max := 1.0, [61].log_data[35].total := 1629.7471, [61].log_data[35].time := 3600.0, [61].log_data[35].maxminute := 6, [61].log_data[35].valid := 1, [61].log_data[36].max := 1.0, [61].log_data[36].total := 1440.998, [61].log_data[36].time := 3600.0,
        [61].log_data[36].minminute := 4, [61].log_data[36].valid := 1, [61].log_data[37].max := 7.339268, [61].log_data[37].total := 3606.1946, [61].log_data[37].time := 3600.0, [61].log_data[37].maxminute := 21, [61].log_data[37].valid := 1, [61].log_data[38].time := 3600.0, [61].log_data[38].valid := 1, [61].log_data[39].min := 0.99753284, [61].log_data[39].max := 1.02097, [61].log_data[39].total := 3622.211, [61].log_data[39].time := 3600.0, [61].log_data[39].minminute := 23, [61].log_data[39].maxminute := 21, [61].log_data[39].valid := 1, [61].log_data[40].min := 7.5788817, [61].log_data[40].max := 7.5950956, [61].log_data[40].total := 27321.082, [61].log_data[40].time := 3600.0, [61].log_data[40].minminute := 58, [61].log_data[40].maxminute := 40, [61].log_data[40].valid := 1, [61].log_data[41].min := 0.022932617, [61].log_data[41].max := 0.037458252, [61].log_data[41].total := 92.38358, [61].log_data[41].time := 3600.0, [61].log_data[41].minminute := 1, [61].log_data[41].maxminute := 19, [61].log_data[41].valid := 1, [61].log_data[42].min := 2.2917604, [61].log_data[42].max := 2.296707, [61].log_data[42].total := 8260.343, [61].log_data[42].time := 3600.0, [61].log_data[42].minminute := 25, [61].log_data[42].maxminute := 8, [61].log_data[42].valid := 1, [61].log_data[43].min := -0.27999878, [61].log_data[43].max := -0.26000214, [61].log_data[43].total := -987.4656, [61].log_data[43].time := 3600.0, [61].log_data[43].maxminute := 2, [61].log_data[43].valid := 1, [61].log_data[44].min := -0.3199997, [61].log_data[44].max := -0.30000305, [61].log_data[44].total := -1080.8656, [61].log_data[44].time := 3600.0, [61].log_data[44].valid := 1, [61].log_data[45].time := 3600.0, [61].log_data[45].valid := 1, [61].log_data[46].time := 3600.0, [61].log_data[46].valid := 1, [61].log_data[47].time := 3600.0, [61].log_data[47].valid := 1, [61].log_data[48].min := 6.5890236, [61].log_data[48].max := 6.981998, [61].log_data[48].total := 24248.922, [61].log_data[48].time := 3600.0, [61].log_data[48].minminute := 54, [61].log_data[48].maxminute := 26,
        [61].log_data[48].valid := 1, [61].log_data[49].min := 7.027787, [61].log_data[49].max := 9.678309, [61].log_data[49].total := 30298.229, [61].log_data[49].time := 3600.0, [61].log_data[49].minminute := 50, [61].log_data[49].maxminute := 21, [61].log_data[49].valid := 1, [61].log_data[50].min := 2.1121538, [61].log_data[50].max := 2.2253356, [61].log_data[50].total := 7829.6333, [61].log_data[50].time := 3600.0, [61].log_data[50].minminute := 21, [61].log_data[50].maxminute := 28, [61].log_data[50].valid := 1, [61].log_data[51].time := 3600.0, [61].log_data[51].valid := 1, [61].log_data[52].min := -3.0800018, [61].log_data[52].max := 0.11999512, [61].log_data[52].total := -7606.842, [61].log_data[52].time := 3600.0, [61].log_data[52].minminute := 2, [61].log_data[52].valid := 1, [61].log_data[53].min := -2.5200043, [61].log_data[53].max := 0.27999878, [61].log_data[53].total := -7122.1816, [61].log_data[53].time := 3600.0, [61].log_data[53].minminute := 22, [61].log_data[53].maxminute := 26, [61].log_data[53].valid := 1, [61].log_data[54].max := 0.58449996, [61].log_data[54].total := 1217.7056, [61].log_data[54].time := 3600.0, [61].log_data[54].maxminute := 2, [61].log_data[54].valid := 1, [61].log_data[55].max := 0.539, [61].log_data[55].total := 1217.4358, [61].log_data[55].time := 3600.0, [61].log_data[55].minminute := 4, [61].log_data[55].maxminute := 48, [61].log_data[55].valid := 1, [61].log_data[56].min := 0.15993154, [61].log_data[56].max := 0.16040264, [61].log_data[56].total := 576.43243, [61].log_data[56].time := 3600.0, [61].log_data[56].minminute := 59, [61].log_data[56].maxminute := 29, [61].log_data[56].valid := 1, [61].log_data[57].min := 0.26694962, [61].log_data[57].max := 0.26832363, [61].log_data[57].total := 964.8293, [61].log_data[57].time := 3600.0, [61].log_data[57].minminute := 59, [61].log_data[57].maxminute := 2, [61].log_data[57].valid := 1, [61].log_data[58].time := 3600.0, [61].log_data[58].valid := 1, [61].log_data[59].time := 3600.0, [61].log_data[59].valid := 1, [61].log_data[60].valid := 1,
        [61].log_data[61].valid := 1, [61].log_data[62].valid := 1, [61].log_data[63].valid := 1, [61].log_data[64].valid := 1, [61].log_data[65].valid := 1, [61].log_data[66].valid := 1, [61].log_data[67].valid := 1, [61].log_data[68].valid := 1, [61].log_data[69].valid := 1, [61].log_data[70].valid := 1, [61].log_data[71].valid := 1, [61].log_data[72].valid := 1, [61].log_data[73].valid := 1, [61].log_data[74].valid := 1, [61].log_data[75].valid := 1, [61].log_data[76].valid := 1, [61].log_data[77].valid := 1, [61].log_data[78].valid := 1, [61].log_data[79].valid := 1, [61].log_data[80].valid := 1, [61].log_data[81].valid := 1, [61].log_data[82].valid := 1, [61].log_data[83].valid := 1, [61].log_data[84].valid := 1, [61].log_data[85].valid := 1, [61].log_data[86].valid := 1, [61].log_data[87].valid := 1, [61].log_data[88].valid := 1, [61].log_data[89].valid := 1, [61].log_data[90].valid := 1, [61].log_data[91].valid := 1, [61].log_data[92].valid := 1, [61].log_data[93].valid := 1, [61].log_data[94].valid := 1, [61].log_data[95].valid := 1, [61].log_data[96].valid := 1, [61].log_data[97].valid := 1, [61].log_data[98].valid := 1, [61].log_data[99].valid := 1, [61].log_data[100].valid := 1, [61].log_data[101].valid := 1, [61].log_data[102].valid := 1, [61].log_data[103].valid := 1, [61].log_data[104].valid := 1, [61].log_data[105].valid := 1, [61].log_data[106].valid := 1, [61].log_data[107].valid := 1, [61].log_data[108].valid := 1, [61].log_data[109].valid := 1, [61].log_data[110].valid := 1, [61].log_data[111].valid := 1, [61].log_data[112].valid := 1, [61].log_data[113].valid := 1, [61].log_data[114].valid := 1, [61].log_data[115].valid := 1, [61].log_data[116].valid := 1, [61].log_data[117].valid := 1, [61].log_data[118].valid := 1, [61].log_data[119].valid := 1, [61].log_data[120].valid := 1,
        [61].log_data[121].valid := 1, [61].log_data[122].valid := 1, [61].log_data[123].valid := 1, [61].log_data[124].valid := 1, [61].time.Year := 2023, [61].time.Month := 1, [61].time.Day := 15, [61].time.Hour := 16, [61].time.Minute := 59, [61].time.Second := 59, [62].log_data[0].min := 1.0, [62].log_data[0].max := 1.0, [62].log_data[0].total := 3600.0, [62].log_data[0].time := 3600.0, [62].log_data[0].valid := 1, [62].log_data[1].max := 1.0, [62].log_data[1].total := 546.0, [62].log_data[1].time := 3600.0, [62].log_data[1].maxminute := 31, [62].log_data[1].valid := 1, [62].log_data[2].max := 1.0, [62].log_data[2].total := 542.5, [62].log_data[2].time := 3600.0, [62].log_data[2].maxminute := 31, [62].log_data[2].valid := 1, [62].log_data[3].time := 3600.0, [62].log_data[3].valid := 1, [62].log_data[4].time := 3600.0, [62].log_data[4].valid := 1, [62].log_data[5].max := 1.0, [62].log_data[5].total := 238.5, [62].log_data[5].time := 3600.0, [62].log_data[5].maxminute := 33, [62].log_data[5].valid := 1, [62].log_data[6].time := 3600.0, [62].log_data[6].valid := 1, [62].log_data[7].time := 3600.0, [62].log_data[7].valid := 1, [62].log_data[8].min := 1.0, [62].log_data[8].max := 1.0, [62].log_data[8].total := 3600.0, [62].log_data[8].time := 3600.0, [62].log_data[8].valid := 1, [62].log_data[9].min := 1.0, [62].log_data[9].max := 1.0, [62].log_data[9].total := 3600.0, [62].log_data[9].time := 3600.0, [62].log_data[9].valid := 1, [62].log_data[10].min := 1.0, [62].log_data[10].max := 1.0, [62].log_data[10].total := 3600.0, [62].log_data[10].time := 3600.0, [62].log_data[10].valid := 1, [62].log_data[11].time := 3600.0, [62].log_data[11].valid := 1, [62].log_data[12].min := 1.0, [62].log_data[12].max := 1.0, [62].log_data[12].total := 3600.0, [62].log_data[12].time := 3600.0, [62].log_data[12].valid := 1,
        [62].log_data[13].min := 1.0, [62].log_data[13].max := 1.0, [62].log_data[13].total := 3600.0, [62].log_data[13].time := 3600.0, [62].log_data[13].valid := 1, [62].log_data[14].time := 3600.0, [62].log_data[14].valid := 1, [62].log_data[15].time := 3600.0, [62].log_data[15].valid := 1, [62].log_data[16].time := 3600.0, [62].log_data[16].valid := 1, [62].log_data[17].min := 1.0, [62].log_data[17].max := 1.0, [62].log_data[17].total := 3600.0, [62].log_data[17].time := 3600.0, [62].log_data[17].valid := 1, [62].log_data[18].time := 3600.0, [62].log_data[18].valid := 1, [62].log_data[19].time := 3600.0, [62].log_data[19].valid := 1, [62].log_data[20].time := 3600.0, [62].log_data[20].valid := 1, [62].log_data[21].min := 1.0, [62].log_data[21].max := 1.0, [62].log_data[21].total := 3600.0, [62].log_data[21].time := 3600.0, [62].log_data[21].valid := 1, [62].log_data[22].time := 3600.0, [62].log_data[22].valid := 1, [62].log_data[23].time := 3600.0, [62].log_data[23].valid := 1, [62].log_data[24].time := 3600.0, [62].log_data[24].valid := 1, [62].log_data[25].time := 3600.0, [62].log_data[25].valid := 1, [62].log_data[26].time := 3600.0, [62].log_data[26].valid := 1, [62].log_data[27].time := 3600.0, [62].log_data[27].valid := 1, [62].log_data[28].time := 3600.0, [62].log_data[28].valid := 1, [62].log_data[29].min := 1.0, [62].log_data[29].max := 1.0, [62].log_data[29].total := 3600.0, [62].log_data[29].time := 3600.0, [62].log_data[29].valid := 1, [62].log_data[30].min := 1.0, [62].log_data[30].max := 1.0, [62].log_data[30].total := 3600.0, [62].log_data[30].time := 3600.0, [62].log_data[30].valid := 1, [62].log_data[31].max := 1.0, [62].log_data[31].total := 1629.7471, [62].log_data[31].time := 3600.0, [62].log_data[31].maxminute := 5, [62].log_data[31].valid := 1, [62].log_data[32].max := 1.0, [62].log_data[32].total := 1440.998, [62].log_data[32].time := 3600.0, [62].log_data[32].minminute := 3,
        [62].log_data[32].valid := 1, [62].log_data[33].time := 3600.0, [62].log_data[33].valid := 1, [62].log_data[34].time := 3600.0, [62].log_data[34].valid := 1, [62].log_data[35].max := 1.0, [62].log_data[35].total := 1602.2471, [62].log_data[35].time := 3600.0, [62].log_data[35].maxminute := 9, [62].log_data[35].valid := 1, [62].log_data[36].max := 1.0, [62].log_data[36].total := 1556.498, [62].log_data[36].time := 3600.0, [62].log_data[36].minminute := 7, [62].log_data[36].valid := 1, [62].log_data[37].max := 7.504938, [62].log_data[37].total := 3545.084, [62].log_data[37].time := 3600.0, [62].log_data[37].maxminute := 32, [62].log_data[37].valid := 1, [62].log_data[38].time := 3600.0, [62].log_data[38].valid := 1, [62].log_data[39].min := 0.99776834, [62].log_data[39].max := 1.0210879, [62].log_data[39].total := 3620.3164, [62].log_data[39].time := 3600.0, [62].log_data[39].minminute := 39, [62].log_data[39].maxminute := 33, [62].log_data[39].valid := 1, [62].log_data[40].min := 7.583004, [62].log_data[40].max := 7.597843, [62].log_data[40].total := 27323.35, [62].log_data[40].time := 3600.0, [62].log_data[40].minminute := 17, [62].log_data[40].maxminute := 40, [62].log_data[40].valid := 1, [62].log_data[41].min := 0.02273633, [62].log_data[41].max := 0.0384397, [62].log_data[41].total := 91.73066, [62].log_data[41].time := 3600.0, [62].log_data[41].minminute := 31, [62].log_data[41].maxminute := 47, [62].log_data[41].valid := 1, [62].log_data[42].min := 2.2916427, [62].log_data[42].max := 2.2968247, [62].log_data[42].total := 8260.36, [62].log_data[42].time := 3600.0, [62].log_data[42].minminute := 32, [62].log_data[42].maxminute := 39, [62].log_data[42].valid := 1, [62].log_data[43].min := -0.27999878, [62].log_data[43].max := -0.26000214, [62].log_data[43].total := -1007.54156, [62].log_data[43].time := 3600.0, [62].log_data[43].valid := 1, [62].log_data[44].min := -0.3199997, [62].log_data[44].max := -0.30000305, [62].log_data[44].total := -1091.7234, [62].log_data[44].time := 3600.0, [62].log_data[44].valid := 1,
